LIN {X 0.012,Y -514.409,Z 331.146,A 0.000,B 0.000,C 90.000,E1 62.281} C_DIS
LIN {X 0.151,Y -518.654,Z 331.138,A 0.000,B 0.000,C 90.000,E1 60.795} C_DIS
LIN {X 0.232,Y -524.544,Z 331.127,A 0.000,B 0.000,C 90.000,E1 58.742} C_DIS
LIN {X -0.129,Y -529.522,Z 331.117,A 0.000,B 0.000,C 90.000,E1 57.041} C_DIS
LIN {X -0.088,Y -534.347,Z 331.107,A 0.000,B 0.000,C 90.000,E1 55.308} C_DIS
LIN {X 0.036,Y -537.358,Z 331.101,A 0.000,B 0.000,C 90.000,E1 54.149} C_DIS
LIN {X 0.091,Y -540.930,Z 331.093,A 0.000,B 0.000,C 90.000,E1 52.718} C_DIS
LIN {X -0.217,Y -544.110,Z 331.085,A 0.000,B 0.000,C 90.000,E1 51.331} C_DIS
LIN {X -0.125,Y -546.940,Z 331.077,A 0.000,B 0.000,C 90.000,E1 49.908} C_DIS
LIN {X 0.018,Y -549.384,Z 331.069,A 0.000,B 0.000,C 90.000,E1 48.485} C_DIS
LIN {X -0.259,Y -551.029,Z 331.063,A 0.000,B 0.000,C 90.000,E1 47.391} C_DIS
LIN {X -0.155,Y -552.114,Z 331.059,A 0.000,B 0.000,C 90.000,E1 46.539} C_DIS
LIN {X 0.343,Y -552.994,Z 331.054,A 0.000,B 0.000,C 90.000,E1 45.648} C_DIS
LIN {X 0.031,Y -553.500,Z 331.051,A 0.000,B 0.000,C 90.000,E1 45.121} C_DIS
LIN {X -0.195,Y -554.104,Z 331.045,A 0.000,B 0.000,C 90.000,E1 44.028} C_DIS
LIN {X -0.056,Y -554.318,Z 331.040,A 0.000,B 0.000,C 90.000,E1 43.176} C_DIS
LIN {X 0.110,Y -554.396,Z 331.034,A 0.000,B 0.000,C 90.000,E1 42.043} C_DIS
LIN {X -0.045,Y -553.917,Z 331.026,A 0.000,B 0.000,C 90.000,E1 40.663} C_DIS
LIN {X -0.209,Y -553.210,Z 331.020,A 0.000,B 0.000,C 90.000,E1 39.564} C_DIS
LIN {X 0.056,Y -552.229,Z 331.014,A 0.000,B 0.000,C 90.000,E1 38.418} C_DIS
LIN {X 0.062,Y -550.152,Z 331.003,A 0.000,B 0.000,C 90.000,E1 36.457} C_DIS
LIN {X 0.287,Y -548.915,Z 330.996,A 0.000,B 0.000,C 90.000,E1 35.311} C_DIS
LIN {X -0.221,Y -545.981,Z 330.982,A 0.000,B 0.000,C 90.000,E1 32.832} C_DIS
LIN {X 0.076,Y -543.685,Z 330.970,A 0.000,B 0.000,C 90.000,E1 30.541} C_DIS
LIN {X 0.017,Y -541.800,Z 330.959,A 0.000,B 0.000,C 90.000,E1 28.565} C_DIS
LIN {X 0.132,Y -539.961,Z 330.948,A 0.000,B 0.000,C 90.000,E1 26.565} C_DIS
LIN {X -0.042,Y -538.136,Z 330.937,A 0.000,B 0.000,C 90.000,E1 24.591} C_DIS
LIN {X 0.146,Y -535.740,Z 330.921,A 0.000,B 0.000,C 90.000,E1 21.716} C_DIS
LIN {X -0.070,Y -534.402,Z 330.908,A 0.000,B 0.000,C 90.000,E1 19.450} C_DIS
LIN {X 0.083,Y -533.648,Z 330.900,A 0.000,B 0.000,C 90.000,E1 18.000} C_DIS
LIN {X -0.002,Y -532.590,Z 330.886,A 0.000,B 0.000,C 90.000,E1 15.426} C_DIS
LIN {X 0.156,Y -531.870,Z 330.870,A 0.000,B 0.000,C 90.000,E1 12.535} C_DIS
LIN {X -0.064,Y -531.909,Z 330.859,A 0.000,B 0.000,C 90.000,E1 10.546} C_DIS
LIN {X 0.059,Y -532.143,Z 330.851,A 0.000,B 0.000,C 90.000,E1 9.095} C_DIS
LIN {X 0.283,Y -533.157,Z 330.833,A 0.000,B 0.000,C 90.000,E1 5.910} C_DIS
LIN {X -0.208,Y -534.755,Z 330.817,A 0.000,B 0.000,C 90.000,E1 3.094} C_DIS
LIN {X -0.196,Y -536.050,Z 330.808,A 0.000,B 0.000,C 90.000,E1 1.375} C_DIS
LIN {X 0.232,Y -538.074,Z 330.794,A 0.000,B 0.000,C 90.000,E1 358.912} C_DIS
LIN {X -0.140,Y -541.024,Z 330.780,A 0.000,B 0.000,C 90.000,E1 356.388} C_DIS
LIN {X -0.052,Y -542.072,Z 330.775,A 0.000,B 0.000,C 90.000,E1 355.527} C_DIS
LIN {X -0.243,Y -544.870,Z 330.763,A 0.000,B 0.000,C 90.000,E1 353.280} C_DIS
LIN {X -0.073,Y -550.293,Z 330.747,A 0.000,B 0.000,C 90.000,E1 350.443} C_DIS
LIN {X 0.094,Y -554.449,Z 330.736,A 0.000,B 0.000,C 90.000,E1 348.465} C_DIS
LIN {X 0.198,Y -558.087,Z 330.728,A 0.000,B 0.000,C 90.000,E1 347.061} C_DIS
LIN {X -0.196,Y -561.292,Z 330.722,A 0.000,B 0.000,C 90.000,E1 345.992} C_DIS
LIN {X -0.225,Y -565.993,Z 330.713,A 0.000,B 0.000,C 90.000,E1 344.338} C_DIS
LIN {X -0.212,Y -571.858,Z 330.702,A 0.000,B 0.000,C 90.000,E1 342.417} C_DIS
LIN {X -0.063,Y -576.026,Z 330.695,A 0.000,B 0.000,C 90.000,E1 341.040} C_DIS
LIN {X 0.156,Y -579.489,Z 330.689,A 0.000,B 0.000,C 90.000,E1 339.934} C_DIS
LIN {X 0.000,Y -586.299,Z 330.677,A 0.000,B 0.000,C 90.000,E1 337.794} C_DIS
LIN {X 0.140,Y -591.574,Z 330.668,A 0.000,B 0.000,C 90.000,E1 336.177} C_DIS
LIN {X 0.011,Y -598.007,Z 330.657,A 0.000,B 0.000,C 90.000,E1 334.332} C_DIS
LIN {X 0.172,Y -602.682,Z 330.650,A 0.000,B 0.000,C 90.000,E1 332.999} C_DIS
LIN {X 0.099,Y -608.216,Z 330.641,A 0.000,B 0.000,C 90.000,E1 331.435} C_DIS
LIN {X 0.103,Y -614.880,Z 330.631,A 0.000,B 0.000,C 90.000,E1 329.616} C_DIS
LIN {X 0.092,Y -618.751,Z 330.626,A 0.000,B 0.000,C 90.000,E1 328.584} C_DIS
LIN {X -0.186,Y -622.410,Z 330.620,A 0.000,B 0.000,C 90.000,E1 327.582} C_DIS
LIN {X -0.081,Y -625.914,Z 330.614,A 0.000,B 0.000,C 90.000,E1 326.548} C_DIS
LIN {X 0.072,Y -629.105,Z 330.608,A 0.000,B 0.000,C 90.000,E1 325.515} C_DIS
LIN {X -0.253,Y -632.881,Z 330.601,A 0.000,B 0.000,C 90.000,E1 324.276} C_DIS
LIN {X -0.157,Y -636.478,Z 330.594,A 0.000,B 0.000,C 90.000,E1 323.004} C_DIS
LIN {X 0.178,Y -642.080,Z 330.583,A 0.000,B 0.000,C 90.000,E1 320.964} C_DIS
LIN {X 0.162,Y -647.168,Z 330.574,A 0.000,B 0.000,C 90.000,E1 319.218} C_DIS
LIN {X -0.158,Y -651.503,Z 330.565,A 0.000,B 0.000,C 90.000,E1 317.757} C_DIS
LIN {X -0.002,Y -657.646,Z 330.554,A 0.000,B 0.000,C 90.000,E1 315.769} C_DIS
LIN {X 0.352,Y -660.733,Z 330.549,A 0.000,B 0.000,C 90.000,E1 314.757} C_DIS
LIN {X 0.263,Y -665.160,Z 330.541,A 0.000,B 0.000,C 90.000,E1 313.299} C_DIS
LIN {X 0.285,Y -669.342,Z 330.533,A 0.000,B 0.000,C 90.000,E1 311.838} C_DIS
LIN {X 0.379,Y -672.572,Z 330.526,A 0.000,B 0.000,C 90.000,E1 310.620} C_DIS
LIN {X 0.104,Y -676.131,Z 330.518,A 0.000,B 0.000,C 90.000,E1 309.197} C_DIS
LIN {X 0.254,Y -677.790,Z 330.514,A 0.000,B 0.000,C 90.000,E1 308.463} C_DIS
LIN {X 0.021,Y -679.783,Z 330.509,A 0.000,B 0.000,C 90.000,E1 307.523} C_DIS
LIN {X -0.187,Y -681.527,Z 330.503,A 0.000,B 0.000,C 90.000,E1 306.583} C_DIS
LIN {X 0.174,Y -682.972,Z 330.498,A 0.000,B 0.000,C 90.000,E1 305.598} C_DIS
LIN {X -0.007,Y -684.060,Z 330.493,A 0.000,B 0.000,C 90.000,E1 304.659} C_DIS
LIN {X -0.201,Y -684.530,Z 330.490,A 0.000,B 0.000,C 90.000,E1 304.199} C_DIS
LIN {X 0.189,Y -684.919,Z 330.486,A 0.000,B 0.000,C 90.000,E1 303.452} C_DIS
LIN {X 0.011,Y -685.079,Z 330.482,A 0.000,B 0.000,C 90.000,E1 302.752} C_DIS
LIN {X -0.172,Y -684.918,Z 330.478,A 0.000,B 0.000,C 90.000,E1 302.054} C_DIS
LIN {X 0.068,Y -684.319,Z 330.473,A 0.000,B 0.000,C 90.000,E1 301.082} C_DIS
LIN {X -0.136,Y -683.579,Z 330.469,A 0.000,B 0.000,C 90.000,E1 300.384} C_DIS
LIN {X -0.106,Y -682.543,Z 330.465,A 0.000,B 0.000,C 90.000,E1 299.667} C_DIS
LIN {X 0.122,Y -680.896,Z 330.460,A 0.000,B 0.000,C 90.000,E1 298.693} C_DIS
LIN {X 0.131,Y -679.393,Z 330.456,A 0.000,B 0.000,C 90.000,E1 297.975} C_DIS
LIN {X -0.094,Y -676.631,Z 330.449,A 0.000,B 0.000,C 90.000,E1 296.796} C_DIS
LIN {X -0.069,Y -673.699,Z 330.442,A 0.000,B 0.000,C 90.000,E1 295.591} C_DIS
LIN {X -0.088,Y -670.569,Z 330.435,A 0.000,B 0.000,C 90.000,E1 294.387} C_DIS
LIN {X 0.182,Y -667.241,Z 330.429,A 0.000,B 0.000,C 90.000,E1 293.153} C_DIS
LIN {X 0.063,Y -662.413,Z 330.419,A 0.000,B 0.000,C 90.000,E1 291.461} C_DIS
LIN {X -0.038,Y -657.821,Z 330.410,A 0.000,B 0.000,C 90.000,E1 289.758} C_DIS
LIN {X -0.114,Y -654.115,Z 330.402,A 0.000,B 0.000,C 90.000,E1 288.290} C_DIS
LIN {X -0.257,Y -648.922,Z 330.389,A 0.000,B 0.000,C 90.000,E1 286.079} C_DIS
LIN {X 0.199,Y -645.195,Z 330.380,A 0.000,B 0.000,C 90.000,E1 284.300} C_DIS
LIN {X -0.043,Y -639.443,Z 330.362,A 0.000,B 0.000,C 90.000,E1 281.074} C_DIS
LIN {X 0.336,Y -635.832,Z 330.346,A 0.000,B 0.000,C 90.000,E1 278.276} C_DIS
LIN {X 0.019,Y -633.257,Z 330.329,A 0.000,B 0.000,C 90.000,E1 275.277} C_DIS
LIN {X -0.167,Y -631.822,Z 330.311,A 0.000,B 0.000,C 90.000,E1 272.007} C_DIS
LIN {X -0.008,Y -631.589,Z 330.298,A 0.000,B 0.000,C 90.000,E1 269.714} C_DIS
LIN {X 0.147,Y -632.009,Z 330.286,A 0.000,B 0.000,C 90.000,E1 267.421} C_DIS
LIN {X 0.246,Y -632.814,Z 330.276,A 0.000,B 0.000,C 90.000,E1 265.641} C_DIS
LIN {X -0.211,Y -633.900,Z 330.266,A 0.000,B 0.000,C 90.000,E1 263.913} C_DIS
LIN {X 0.258,Y -635.065,Z 330.258,A 0.000,B 0.000,C 90.000,E1 262.356} C_DIS
LIN {X -0.263,Y -636.792,Z 330.247,A 0.000,B 0.000,C 90.000,E1 260.387} C_DIS
LIN {X 0.114,Y -638.970,Z 330.235,A 0.000,B 0.000,C 90.000,E1 258.342} C_DIS
LIN {X 0.081,Y -641.221,Z 330.226,A 0.000,B 0.000,C 90.000,E1 256.589} C_DIS
LIN {X 0.072,Y -642.543,Z 330.220,A 0.000,B 0.000,C 90.000,E1 255.589} C_DIS
LIN {X -0.227,Y -643.320,Z 330.216,A 0.000,B 0.000,C 90.000,E1 254.866} C_DIS
LIN {X -0.186,Y -644.381,Z 330.209,A 0.000,B 0.000,C 90.000,E1 253.614} C_DIS
LIN {X -0.133,Y -645.125,Z 330.202,A 0.000,B 0.000,C 90.000,E1 252.362} C_DIS
LIN {X 0.223,Y -645.400,Z 330.198,A 0.000,B 0.000,C 90.000,E1 251.583} C_DIS
LIN {X -0.033,Y -645.324,Z 330.194,A 0.000,B 0.000,C 90.000,E1 250.859} C_DIS
LIN {X 0.024,Y -645.305,Z 330.192,A 0.000,B 0.000,C 90.000,E1 250.604} C_DIS
LIN {X -0.232,Y -644.846,Z 330.188,A 0.000,B 0.000,C 90.000,E1 249.880} C_DIS
LIN {X -0.332,Y -644.440,Z 330.185,A 0.000,B 0.000,C 90.000,E1 249.390} C_DIS
LIN {X 0.229,Y -643.507,Z 330.181,A 0.000,B 0.000,C 90.000,E1 248.592} C_DIS
LIN {X 0.118,Y -642.776,Z 330.178,A 0.000,B 0.000,C 90.000,E1 248.103} C_DIS
LIN {X 0.064,Y -641.430,Z 330.174,A 0.000,B 0.000,C 90.000,E1 247.358} C_DIS
LIN {X -0.064,Y -640.421,Z 330.172,A 0.000,B 0.000,C 90.000,E1 246.869} C_DIS
LIN {X -0.090,Y -638.024,Z 330.166,A 0.000,B 0.000,C 90.000,E1 245.869} C_DIS
LIN {X 0.069,Y -636.071,Z 330.162,A 0.000,B 0.000,C 90.000,E1 245.101} C_DIS
LIN {X 0.167,Y -634.684,Z 330.159,A 0.000,B 0.000,C 90.000,E1 244.588} C_DIS
LIN {X 0.059,Y -631.483,Z 330.153,A 0.000,B 0.000,C 90.000,E1 243.589} C_DIS
LIN {X 0.179,Y -628.105,Z 330.148,A 0.000,B 0.000,C 90.000,E1 242.564} C_DIS
LIN {X 0.007,Y -623.774,Z 330.141,A 0.000,B 0.000,C 90.000,E1 241.307} C_DIS
LIN {X 0.015,Y -620.333,Z 330.135,A 0.000,B 0.000,C 90.000,E1 240.284} C_DIS
LIN {X 0.010,Y -615.064,Z 330.126,A 0.000,B 0.000,C 90.000,E1 238.742} C_DIS
LIN {X 0.231,Y -609.789,Z 330.118,A 0.000,B 0.000,C 90.000,E1 237.168} C_DIS
LIN {X 0.082,Y -605.275,Z 330.111,A 0.000,B 0.000,C 90.000,E1 235.881} C_DIS
LIN {X 0.083,Y -597.989,Z 330.099,A 0.000,B 0.000,C 90.000,E1 233.783} C_DIS
LIN {X -0.292,Y -594.305,Z 330.093,A 0.000,B 0.000,C 90.000,E1 232.763} C_DIS
LIN {X 0.108,Y -586.649,Z 330.081,A 0.000,B 0.000,C 90.000,E1 230.598} C_DIS
LIN {X 0.131,Y -582.072,Z 330.074,A 0.000,B 0.000,C 90.000,E1 229.256} C_DIS
LIN {X 0.029,Y -574.882,Z 330.062,A 0.000,B 0.000,C 90.000,E1 227.106} C_DIS
LIN {X 0.197,Y -570.377,Z 330.054,A 0.000,B 0.000,C 90.000,E1 225.729} C_DIS
LIN {X -0.018,Y -565.003,Z 330.045,A 0.000,B 0.000,C 90.000,E1 224.109} C_DIS
LIN {X 0.140,Y -558.793,Z 330.034,A 0.000,B 0.000,C 90.000,E1 222.162} C_DIS
LIN {X -0.225,Y -552.620,Z 330.024,A 0.000,B 0.000,C 90.000,E1 220.253} C_DIS
LIN {X 0.053,Y -547.411,Z 330.014,A 0.000,B 0.000,C 90.000,E1 218.543} C_DIS
LIN {X -0.096,Y -541.470,Z 330.003,A 0.000,B 0.000,C 90.000,E1 216.583} C_DIS
LIN {X 0.168,Y -535.054,Z 329.991,A 0.000,B 0.000,C 90.000,E1 214.278} C_DIS
LIN {X -0.052,Y -529.022,Z 329.978,A 0.000,B 0.000,C 90.000,E1 212.005} C_DIS
LIN {X -0.233,Y -524.175,Z 329.967,A 0.000,B 0.000,C 90.000,E1 210.001} C_DIS
LIN {X -0.078,Y -521.442,Z 329.960,A 0.000,B 0.000,C 90.000,E1 208.821} C_DIS
LIN {X 0.200,Y -516.746,Z 329.949,A 0.000,B 0.000,C 90.000,E1 206.744} C_DIS
LIN {X 0.123,Y -513.496,Z 329.941,A 0.000,B 0.000,C 90.000,E1 205.283} C_DIS
LIN {X -0.126,Y -510.935,Z 329.934,A 0.000,B 0.000,C 90.000,E1 204.131} C_DIS
LIN {X -0.055,Y -507.615,Z 329.926,A 0.000,B 0.000,C 90.000,E1 202.642} C_DIS
LIN {X -0.052,Y -502.946,Z 329.914,A 0.000,B 0.000,C 90.000,E1 200.556} C_DIS
LIN {X 0.233,Y -498.998,Z 329.904,A 0.000,B 0.000,C 90.000,E1 198.725} C_DIS
LIN {X 0.258,Y -495.156,Z 329.894,A 0.000,B 0.000,C 90.000,E1 196.913} C_DIS
LIN {X -0.085,Y -491.558,Z 329.884,A 0.000,B 0.000,C 90.000,E1 195.134} C_DIS
LIN {X -0.023,Y -488.185,Z 329.874,A 0.000,B 0.000,C 90.000,E1 193.300} C_DIS
LIN {X -0.030,Y -485.458,Z 329.865,A 0.000,B 0.000,C 90.000,E1 191.771} C_DIS
LIN {X -0.188,Y -482.775,Z 329.857,A 0.000,B 0.000,C 90.000,E1 190.254} C_DIS
LIN {X -0.145,Y -479.614,Z 329.847,A 0.000,B 0.000,C 90.000,E1 188.398} C_DIS
LIN {X -0.090,Y -475.772,Z 329.833,A 0.000,B 0.000,C 90.000,E1 185.910} C_DIS
LIN {X 0.177,Y -472.347,Z 329.819,A 0.000,B 0.000,C 90.000,E1 183.383} C_DIS
LIN {X -0.153,Y -469.340,Z 329.805,A 0.000,B 0.000,C 90.000,E1 180.917} C_DIS
LIN {X -0.126,Y -467.003,Z 329.791,A 0.000,B 0.000,C 90.000,E1 178.396} C_DIS
LIN {X 0.107,Y -464.884,Z 329.772,A 0.000,B 0.000,C 90.000,E1 174.894} C_DIS
LIN {X -0.050,Y -464.115,Z 329.756,A 0.000,B 0.000,C 90.000,E1 172.064} C_DIS
LIN {X -0.148,Y -464.067,Z 329.744,A 0.000,B 0.000,C 90.000,E1 169.859} C_DIS
LIN {X 0.200,Y -465.056,Z 329.721,A 0.000,B 0.000,C 90.000,E1 165.700} C_DIS
LIN {X 0.061,Y -466.232,Z 329.708,A 0.000,B 0.000,C 90.000,E1 163.504} C_DIS
LIN {X 0.191,Y -469.670,Z 329.686,A 0.000,B 0.000,C 90.000,E1 159.390} C_DIS
LIN {X -0.222,Y -473.534,Z 329.668,A 0.000,B 0.000,C 90.000,E1 156.305} C_DIS
LIN {X 0.131,Y -477.489,Z 329.654,A 0.000,B 0.000,C 90.000,E1 153.768} C_DIS
LIN {X -0.019,Y -482.266,Z 329.641,A 0.000,B 0.000,C 90.000,E1 151.307} C_DIS
LIN {X -0.031,Y -486.993,Z 329.629,A 0.000,B 0.000,C 90.000,E1 149.154} C_DIS
LIN {X 0.089,Y -489.890,Z 329.622,A 0.000,B 0.000,C 90.000,E1 147.916} C_DIS
LIN {X -0.002,Y -493.123,Z 329.615,A 0.000,B 0.000,C 90.000,E1 146.707} C_DIS
LIN {X -0.191,Y -498.875,Z 329.603,A 0.000,B 0.000,C 90.000,E1 144.609} C_DIS
LIN {X 0.180,Y -503.920,Z 329.593,A 0.000,B 0.000,C 90.000,E1 142.763} C_DIS
LIN {X -0.255,Y -507.135,Z 329.587,A 0.000,B 0.000,C 90.000,E1 141.618} C_DIS
LIN {X -0.237,Y -509.324,Z 329.582,A 0.000,B 0.000,C 90.000,E1 140.723} C_DIS
LIN {X -0.192,Y -511.355,Z 329.577,A 0.000,B 0.000,C 90.000,E1 139.828} C_DIS
LIN {X 0.041,Y -514.326,Z 329.569,A 0.000,B 0.000,C 90.000,E1 138.324} C_DIS
LIN {X -0.248,Y -515.862,Z 329.564,A 0.000,B 0.000,C 90.000,E1 137.472} C_DIS
LIN {X 0.209,Y -517.062,Z 329.559,A 0.000,B 0.000,C 90.000,E1 136.539} C_DIS
LIN {X 0.305,Y -517.835,Z 329.554,A 0.000,B 0.000,C 90.000,E1 135.648} C_DIS
LIN {X -0.038,Y -518.443,Z 329.547,A 0.000,B 0.000,C 90.000,E1 134.514} C_DIS
LIN {X 0.075,Y -518.571,Z 329.542,A 0.000,B 0.000,C 90.000,E1 133.623} C_DIS
LIN {X -0.097,Y -518.502,Z 329.539,A 0.000,B 0.000,C 90.000,E1 133.056} C_DIS
LIN {X 0.042,Y -518.148,Z 329.534,A 0.000,B 0.000,C 90.000,E1 132.162} C_DIS
LIN {X -0.204,Y -517.471,Z 329.529,A 0.000,B 0.000,C 90.000,E1 131.310} C_DIS
LIN {X -0.066,Y -516.523,Z 329.525,A 0.000,B 0.000,C 90.000,E1 130.415} C_DIS
LIN {X 0.320,Y -515.023,Z 329.518,A 0.000,B 0.000,C 90.000,E1 129.197} C_DIS
LIN {X 0.199,Y -512.590,Z 329.508,A 0.000,B 0.000,C 90.000,E1 127.443} C_DIS
LIN {X -0.120,Y -510.914,Z 329.502,A 0.000,B 0.000,C 90.000,E1 126.297} C_DIS
LIN {X -0.049,Y -509.074,Z 329.495,A 0.000,B 0.000,C 90.000,E1 125.105} C_DIS
LIN {X -0.008,Y -506.958,Z 329.488,A 0.000,B 0.000,C 90.000,E1 123.913} C_DIS
LIN {X 0.034,Y -504.105,Z 329.480,A 0.000,B 0.000,C 90.000,E1 122.418} C_DIS
LIN {X -0.157,Y -502.292,Z 329.475,A 0.000,B 0.000,C 90.000,E1 121.544} C_DIS
LIN {X -0.167,Y -498.590,Z 329.465,A 0.000,B 0.000,C 90.000,E1 119.745} C_DIS
LIN {X -0.108,Y -495.312,Z 329.457,A 0.000,B 0.000,C 90.000,E1 118.231} C_DIS
LIN {X -0.066,Y -490.773,Z 329.445,A 0.000,B 0.000,C 90.000,E1 116.104} C_DIS
LIN {X -0.165,Y -487.434,Z 329.437,A 0.000,B 0.000,C 90.000,E1 114.591} C_DIS
LIN {X 0.121,Y -483.973,Z 329.428,A 0.000,B 0.000,C 90.000,E1 113.025} C_DIS
LIN {X 0.151,Y -479.763,Z 329.418,A 0.000,B 0.000,C 90.000,E1 111.173} C_DIS
LIN {X 0.128,Y -477.600,Z 329.413,A 0.000,B 0.000,C 90.000,E1 110.248} C_DIS
LIN {X -0.134,Y -473.705,Z 329.404,A 0.000,B 0.000,C 90.000,E1 108.725} C_DIS
LIN {X 0.019,Y -470.581,Z 329.397,A 0.000,B 0.000,C 90.000,E1 107.457} C_DIS
LIN {X -0.016,Y -467.271,Z 329.390,A 0.000,B 0.000,C 90.000,E1 106.205} C_DIS
LIN {X 0.118,Y -465.868,Z 329.387,A 0.000,B 0.000,C 90.000,E1 105.662} C_DIS
LIN {X 0.078,Y -465.863,Z 329.387,A 0.000,B 0.000,C 90.000,E1 105.662} C_DIS
LIN {X -0.099,Y -467.672,Z 329.383,A 0.000,B 0.000,C 90.000,E1 104.954} C_DIS
LIN {X -0.141,Y -475.886,Z 329.357,A 0.000,B 0.000,C 90.000,E1 100.254} C_DIS
LIN {X 0.166,Y -476.343,Z 329.355,A 0.000,B 0.000,C 90.000,E1 99.905} C_DIS
LIN {X 0.123,Y -481.853,Z 329.331,A 0.000,B 0.000,C 90.000,E1 95.568} C_DIS
LIN {X -0.031,Y -482.187,Z 329.329,A 0.000,B 0.000,C 90.000,E1 95.277} C_DIS
LIN {X -0.097,Y -485.350,Z 329.305,A 0.000,B 0.000,C 90.000,E1 90.974} C_DIS
LIN {X 0.213,Y -485.533,Z 329.304,A 0.000,B 0.000,C 90.000,E1 90.630} C_DIS
LIN {X -0.065,Y -486.339,Z 329.282,A 0.000,B 0.000,C 90.000,E1 86.674} C_DIS
LIN {X 0.069,Y -486.277,Z 329.278,A 0.000,B 0.000,C 90.000,E1 86.045} C_DIS
LIN {X -0.211,Y -484.694,Z 329.254,A 0.000,B 0.000,C 90.000,E1 81.781} C_DIS
LIN {X 0.137,Y -484.551,Z 329.253,A 0.000,B 0.000,C 90.000,E1 81.432} C_DIS
LIN {X 0.007,Y -480.491,Z 329.227,A 0.000,B 0.000,C 90.000,E1 76.825} C_DIS
LIN {X 0.206,Y -477.337,Z 329.215,A 0.000,B 0.000,C 90.000,E1 74.755} C_DIS
LIN {X 0.166,Y -477.338,Z 329.215,A 0.000,B 0.000,C 90.000,E1 74.755} C_DIS
LIN {X -0.103,Y -480.709,Z 329.210,A 0.000,B 0.000,C 90.000,E1 73.740} C_DIS
LIN {X 0.178,Y -483.615,Z 329.204,A 0.000,B 0.000,C 90.000,E1 72.779} C_DIS
LIN {X -0.100,Y -487.983,Z 329.196,A 0.000,B 0.000,C 90.000,E1 71.275} C_DIS
LIN {X -0.140,Y -492.281,Z 329.187,A 0.000,B 0.000,C 90.000,E1 69.752} C_DIS
LIN {X -0.104,Y -496.633,Z 329.179,A 0.000,B 0.000,C 90.000,E1 68.230} C_DIS
LIN {X 0.125,Y -500.116,Z 329.172,A 0.000,B 0.000,C 90.000,E1 66.997} C_DIS
LIN {X -0.075,Y -506.113,Z 329.161,A 0.000,B 0.000,C 90.000,E1 64.921} C_DIS
LIN {X 0.002,Y -511.279,Z 329.151,A 0.000,B 0.000,C 90.000,E1 63.127} C_DIS
LIN {X -0.264,Y -516.377,Z 329.141,A 0.000,B 0.000,C 90.000,E1 61.385} C_DIS
LIN {X 0.157,Y -520.579,Z 329.133,A 0.000,B 0.000,C 90.000,E1 59.871} C_DIS
LIN {X 0.208,Y -524.782,Z 329.125,A 0.000,B 0.000,C 90.000,E1 58.408} C_DIS
LIN {X -0.149,Y -529.790,Z 329.115,A 0.000,B 0.000,C 90.000,E1 56.707} C_DIS
LIN {X -0.099,Y -533.800,Z 329.107,A 0.000,B 0.000,C 90.000,E1 55.261} C_DIS
LIN {X -0.110,Y -536.848,Z 329.101,A 0.000,B 0.000,C 90.000,E1 54.116} C_DIS
LIN {X -0.070,Y -539.716,Z 329.094,A 0.000,B 0.000,C 90.000,E1 52.970} C_DIS
LIN {X 0.036,Y -542.959,Z 329.086,A 0.000,B 0.000,C 90.000,E1 51.537} C_DIS
LIN {X -0.269,Y -545.289,Z 329.080,A 0.000,B 0.000,C 90.000,E1 50.436} C_DIS
LIN {X 0.184,Y -546.922,Z 329.075,A 0.000,B 0.000,C 90.000,E1 49.542} C_DIS
LIN {X -0.126,Y -548.880,Z 329.069,A 0.000,B 0.000,C 90.000,E1 48.447} C_DIS
LIN {X 0.002,Y -550.532,Z 329.063,A 0.000,B 0.000,C 90.000,E1 47.310} C_DIS
LIN {X 0.102,Y -551.631,Z 329.058,A 0.000,B 0.000,C 90.000,E1 46.458} C_DIS
LIN {X -0.187,Y -552.538,Z 329.054,A 0.000,B 0.000,C 90.000,E1 45.648} C_DIS
LIN {X -0.074,Y -553.249,Z 329.049,A 0.000,B 0.000,C 90.000,E1 44.798} C_DIS
LIN {X 0.048,Y -553.721,Z 329.044,A 0.000,B 0.000,C 90.000,E1 43.947} C_DIS
LIN {X 0.182,Y -553.999,Z 329.040,A 0.000,B 0.000,C 90.000,E1 43.095} C_DIS
LIN {X -0.026,Y -554.142,Z 329.033,A 0.000,B 0.000,C 90.000,E1 42.000} C_DIS
LIN {X 0.178,Y -553.931,Z 329.027,A 0.000,B 0.000,C 90.000,E1 40.862} C_DIS
LIN {X 0.312,Y -553.581,Z 329.023,A 0.000,B 0.000,C 90.000,E1 40.011} C_DIS
LIN {X 0.149,Y -552.782,Z 329.016,A 0.000,B 0.000,C 90.000,E1 38.910} C_DIS
LIN {X -0.087,Y -552.007,Z 329.012,A 0.000,B 0.000,C 90.000,E1 38.096} C_DIS
LIN {X -0.157,Y -550.296,Z 329.002,A 0.000,B 0.000,C 90.000,E1 36.423} C_DIS
LIN {X -0.256,Y -549.056,Z 328.996,A 0.000,B 0.000,C 90.000,E1 35.311} C_DIS
LIN {X -0.002,Y -546.142,Z 328.982,A 0.000,B 0.000,C 90.000,E1 32.752} C_DIS
LIN {X 0.292,Y -543.860,Z 328.969,A 0.000,B 0.000,C 90.000,E1 30.463} C_DIS
LIN {X 0.230,Y -541.988,Z 328.958,A 0.000,B 0.000,C 90.000,E1 28.487} C_DIS
LIN {X -0.142,Y -540.147,Z 328.947,A 0.000,B 0.000,C 90.000,E1 26.539} C_DIS
LIN {X 0.163,Y -538.318,Z 328.936,A 0.000,B 0.000,C 90.000,E1 24.515} C_DIS
LIN {X 0.144,Y -535.937,Z 328.920,A 0.000,B 0.000,C 90.000,E1 21.663} C_DIS
LIN {X -0.084,Y -534.755,Z 328.909,A 0.000,B 0.000,C 90.000,E1 19.685} C_DIS
LIN {X 0.102,Y -533.848,Z 328.900,A 0.000,B 0.000,C 90.000,E1 17.946} C_DIS
LIN {X 0.031,Y -532.786,Z 328.885,A 0.000,B 0.000,C 90.000,E1 15.371} C_DIS
LIN {X 0.202,Y -532.082,Z 328.870,A 0.000,B 0.000,C 90.000,E1 12.479} C_DIS
LIN {X -0.009,Y -532.119,Z 328.858,A 0.000,B 0.000,C 90.000,E1 10.489} C_DIS
LIN {X 0.204,Y -532.355,Z 328.850,A 0.000,B 0.000,C 90.000,E1 9.029} C_DIS
LIN {X -0.210,Y -533.275,Z 328.834,A 0.000,B 0.000,C 90.000,E1 6.201} C_DIS
LIN {X -0.124,Y -534.985,Z 328.817,A 0.000,B 0.000,C 90.000,E1 3.037} C_DIS
LIN {X -0.102,Y -536.507,Z 328.806,A 0.000,B 0.000,C 90.000,E1 1.031} C_DIS
LIN {X -0.211,Y -540.025,Z 328.785,A 0.000,B 0.000,C 90.000,E1 357.249} C_DIS
LIN {X -0.048,Y -542.041,Z 328.775,A 0.000,B 0.000,C 90.000,E1 355.527} C_DIS
LIN {X -0.158,Y -545.172,Z 328.761,A 0.000,B 0.000,C 90.000,E1 352.989} C_DIS
LIN {X -0.077,Y -550.039,Z 328.747,A 0.000,B 0.000,C 90.000,E1 350.443} C_DIS
LIN {X 0.208,Y -554.848,Z 328.734,A 0.000,B 0.000,C 90.000,E1 348.173} C_DIS
LIN {X 0.182,Y -557.700,Z 328.728,A 0.000,B 0.000,C 90.000,E1 347.061} C_DIS
LIN {X 0.183,Y -560.145,Z 328.724,A 0.000,B 0.000,C 90.000,E1 346.228} C_DIS
LIN {X 0.059,Y -566.428,Z 328.711,A 0.000,B 0.000,C 90.000,E1 344.031} C_DIS
LIN {X 0.293,Y -571.413,Z 328.702,A 0.000,B 0.000,C 90.000,E1 342.362} C_DIS
LIN {X -0.109,Y -575.583,Z 328.695,A 0.000,B 0.000,C 90.000,E1 341.040} C_DIS
LIN {X -0.258,Y -579.814,Z 328.687,A 0.000,B 0.000,C 90.000,E1 339.699} C_DIS
LIN {X 0.097,Y -588.430,Z 328.672,A 0.000,B 0.000,C 90.000,E1 336.975} C_DIS
LIN {X 0.006,Y -596.584,Z 328.659,A 0.000,B 0.000,C 90.000,E1 334.588} C_DIS
LIN {X 0.141,Y -601.287,Z 328.652,A 0.000,B 0.000,C 90.000,E1 333.256} C_DIS
LIN {X -0.065,Y -604.086,Z 328.647,A 0.000,B 0.000,C 90.000,E1 332.487} C_DIS
LIN {X -0.160,Y -610.567,Z 328.637,A 0.000,B 0.000,C 90.000,E1 330.667} C_DIS
LIN {X 0.256,Y -615.401,Z 328.630,A 0.000,B 0.000,C 90.000,E1 329.331} C_DIS
LIN {X -0.064,Y -619.250,Z 328.624,A 0.000,B 0.000,C 90.000,E1 328.329} C_DIS
LIN {X -0.005,Y -622.834,Z 328.618,A 0.000,B 0.000,C 90.000,E1 327.296} C_DIS
LIN {X 0.295,Y -625.460,Z 328.614,A 0.000,B 0.000,C 90.000,E1 326.501} C_DIS
LIN {X -0.087,Y -629.421,Z 328.607,A 0.000,B 0.000,C 90.000,E1 325.261} C_DIS
LIN {X -0.046,Y -633.157,Z 328.600,A 0.000,B 0.000,C 90.000,E1 323.989} C_DIS
LIN {X 0.057,Y -636.018,Z 328.594,A 0.000,B 0.000,C 90.000,E1 322.970} C_DIS
LIN {X -0.003,Y -640.931,Z 328.585,A 0.000,B 0.000,C 90.000,E1 321.215} C_DIS
LIN {X -0.032,Y -646.699,Z 328.573,A 0.000,B 0.000,C 90.000,E1 319.218} C_DIS
LIN {X -0.305,Y -650.323,Z 328.567,A 0.000,B 0.000,C 90.000,E1 318.000} C_DIS
LIN {X 0.238,Y -657.144,Z 328.554,A 0.000,B 0.000,C 90.000,E1 315.729} C_DIS
LIN {X 0.126,Y -660.231,Z 328.549,A 0.000,B 0.000,C 90.000,E1 314.757} C_DIS
LIN {X 0.025,Y -664.624,Z 328.541,A 0.000,B 0.000,C 90.000,E1 313.299} C_DIS
LIN {X 0.035,Y -668.772,Z 328.533,A 0.000,B 0.000,C 90.000,E1 311.838} C_DIS
LIN {X 0.118,Y -671.947,Z 328.526,A 0.000,B 0.000,C 90.000,E1 310.620} C_DIS
LIN {X -0.170,Y -675.435,Z 328.518,A 0.000,B 0.000,C 90.000,E1 309.197} C_DIS
LIN {X -0.029,Y -677.057,Z 328.514,A 0.000,B 0.000,C 90.000,E1 308.463} C_DIS
LIN {X 0.284,Y -679.487,Z 328.507,A 0.000,B 0.000,C 90.000,E1 307.237} C_DIS
LIN {X 0.071,Y -681.117,Z 328.502,A 0.000,B 0.000,C 90.000,E1 306.297} C_DIS
LIN {X -0.140,Y -682.177,Z 328.498,A 0.000,B 0.000,C 90.000,E1 305.598} C_DIS
LIN {X -0.340,Y -682.973,Z 328.494,A 0.000,B 0.000,C 90.000,E1 304.898} C_DIS
LIN {X 0.417,Y -683.609,Z 328.490,A 0.000,B 0.000,C 90.000,E1 304.119} C_DIS
LIN {X -0.154,Y -684.005,Z 328.484,A 0.000,B 0.000,C 90.000,E1 303.214} C_DIS
LIN {X -0.338,Y -684.067,Z 328.482,A 0.000,B 0.000,C 90.000,E1 302.752} C_DIS
LIN {X -0.151,Y -684.005,Z 328.479,A 0.000,B 0.000,C 90.000,E1 302.260} C_DIS
LIN {X 0.431,Y -683.409,Z 328.474,A 0.000,B 0.000,C 90.000,E1 301.258} C_DIS
LIN {X -0.132,Y -682.737,Z 328.470,A 0.000,B 0.000,C 90.000,E1 300.590} C_DIS
LIN {X 0.094,Y -681.380,Z 328.465,A 0.000,B 0.000,C 90.000,E1 299.617} C_DIS
LIN {X 0.110,Y -680.120,Z 328.461,A 0.000,B 0.000,C 90.000,E1 298.899} C_DIS
LIN {X -0.286,Y -678.136,Z 328.455,A 0.000,B 0.000,C 90.000,E1 297.975} C_DIS
LIN {X 0.074,Y -675.355,Z 328.449,A 0.000,B 0.000,C 90.000,E1 296.744} C_DIS
LIN {X 0.084,Y -672.367,Z 328.442,A 0.000,B 0.000,C 90.000,E1 295.540} C_DIS
LIN {X 0.210,Y -668.566,Z 328.434,A 0.000,B 0.000,C 90.000,E1 294.079} C_DIS
LIN {X -0.163,Y -665.175,Z 328.427,A 0.000,B 0.000,C 90.000,E1 292.898} C_DIS
LIN {X 0.157,Y -661.049,Z 328.419,A 0.000,B 0.000,C 90.000,E1 291.408} C_DIS
LIN {X 0.032,Y -656.461,Z 328.410,A 0.000,B 0.000,C 90.000,E1 289.704} C_DIS
LIN {X -0.193,Y -652.157,Z 328.400,A 0.000,B 0.000,C 90.000,E1 288.000} C_DIS
LIN {X -0.240,Y -647.587,Z 328.389,A 0.000,B 0.000,C 90.000,E1 286.024} C_DIS
LIN {X -0.259,Y -642.409,Z 328.375,A 0.000,B 0.000,C 90.000,E1 283.536} C_DIS
LIN {X 0.015,Y -637.091,Z 328.357,A 0.000,B 0.000,C 90.000,E1 280.254} C_DIS
LIN {X -0.137,Y -632.935,Z 328.336,A 0.000,B 0.000,C 90.000,E1 276.486} C_DIS
LIN {X 0.098,Y -631.421,Z 328.323,A 0.000,B 0.000,C 90.000,E1 274.188} C_DIS
LIN {X 0.269,Y -630.607,Z 328.311,A 0.000,B 0.000,C 90.000,E1 271.892} C_DIS
LIN {X -0.239,Y -630.394,Z 328.298,A 0.000,B 0.000,C 90.000,E1 269.656} C_DIS
LIN {X -0.120,Y -630.849,Z 328.285,A 0.000,B 0.000,C 90.000,E1 267.364} C_DIS
LIN {X -0.323,Y -631.834,Z 328.274,A 0.000,B 0.000,C 90.000,E1 265.355} C_DIS
LIN {X -0.183,Y -632.982,Z 328.264,A 0.000,B 0.000,C 90.000,E1 263.571} C_DIS
LIN {X 0.342,Y -634.210,Z 328.256,A 0.000,B 0.000,C 90.000,E1 262.008} C_DIS
LIN {X -0.016,Y -635.789,Z 328.246,A 0.000,B 0.000,C 90.000,E1 260.274} C_DIS
LIN {X -0.126,Y -637.726,Z 328.236,A 0.000,B 0.000,C 90.000,E1 258.522} C_DIS
LIN {X -0.047,Y -640.000,Z 328.226,A 0.000,B 0.000,C 90.000,E1 256.756} C_DIS
LIN {X -0.223,Y -641.661,Z 328.219,A 0.000,B 0.000,C 90.000,E1 255.519} C_DIS
LIN {X -0.228,Y -642.720,Z 328.214,A 0.000,B 0.000,C 90.000,E1 254.519} C_DIS
LIN {X -0.052,Y -643.574,Z 328.208,A 0.000,B 0.000,C 90.000,E1 253.504} C_DIS
LIN {X 0.175,Y -644.386,Z 328.201,A 0.000,B 0.000,C 90.000,E1 252.236} C_DIS
LIN {X -0.133,Y -644.663,Z 328.199,A 0.000,B 0.000,C 90.000,E1 251.764} C_DIS
LIN {X 0.265,Y -644.674,Z 328.193,A 0.000,B 0.000,C 90.000,E1 250.732} C_DIS
LIN {X 0.106,Y -644.667,Z 328.192,A 0.000,B 0.000,C 90.000,E1 250.496} C_DIS
LIN {X -0.103,Y -644.105,Z 328.186,A 0.000,B 0.000,C 90.000,E1 249.518} C_DIS
LIN {X -0.209,Y -643.656,Z 328.183,A 0.000,B 0.000,C 90.000,E1 249.028} C_DIS
LIN {X -0.256,Y -642.787,Z 328.179,A 0.000,B 0.000,C 90.000,E1 248.284} C_DIS
LIN {X -0.370,Y -642.034,Z 328.177,A 0.000,B 0.000,C 90.000,E1 247.794} C_DIS
LIN {X 0.158,Y -640.673,Z 328.172,A 0.000,B 0.000,C 90.000,E1 246.997} C_DIS
LIN {X 0.277,Y -639.621,Z 328.170,A 0.000,B 0.000,C 90.000,E1 246.485} C_DIS
LIN {X 0.189,Y -637.822,Z 328.165,A 0.000,B 0.000,C 90.000,E1 245.741} C_DIS
LIN {X 0.396,Y -635.171,Z 328.160,A 0.000,B 0.000,C 90.000,E1 244.717} C_DIS
LIN {X -0.274,Y -632.042,Z 328.154,A 0.000,B 0.000,C 90.000,E1 243.768} C_DIS
LIN {X -0.139,Y -628.709,Z 328.149,A 0.000,B 0.000,C 90.000,E1 242.743} C_DIS
LIN {X -0.055,Y -625.308,Z 328.143,A 0.000,B 0.000,C 90.000,E1 241.719} C_DIS
LIN {X -0.269,Y -620.164,Z 328.134,A 0.000,B 0.000,C 90.000,E1 240.205} C_DIS
LIN {X -0.269,Y -614.975,Z 328.126,A 0.000,B 0.000,C 90.000,E1 238.663} C_DIS
LIN {X 0.191,Y -610.649,Z 328.119,A 0.000,B 0.000,C 90.000,E1 237.327} C_DIS
LIN {X 0.119,Y -607.153,Z 328.113,A 0.000,B 0.000,C 90.000,E1 236.294} C_DIS
LIN {X -0.074,Y -600.861,Z 328.103,A 0.000,B 0.000,C 90.000,E1 234.482} C_DIS
LIN {X 0.068,Y -597.290,Z 328.097,A 0.000,B 0.000,C 90.000,E1 233.417} C_DIS
LIN {X 0.157,Y -593.526,Z 328.091,A 0.000,B 0.000,C 90.000,E1 232.351} C_DIS
LIN {X -0.011,Y -584.202,Z 328.076,A 0.000,B 0.000,C 90.000,E1 229.703} C_DIS
LIN {X -0.326,Y -576.122,Z 328.063,A 0.000,B 0.000,C 90.000,E1 227.310} C_DIS
LIN {X 0.285,Y -571.690,Z 328.055,A 0.000,B 0.000,C 90.000,E1 225.891} C_DIS
LIN {X -0.213,Y -565.387,Z 328.045,A 0.000,B 0.000,C 90.000,E1 224.028} C_DIS
LIN {X -0.128,Y -560.106,Z 328.035,A 0.000,B 0.000,C 90.000,E1 222.366} C_DIS
LIN {X -0.117,Y -554.864,Z 328.026,A 0.000,B 0.000,C 90.000,E1 220.701} C_DIS
LIN {X 0.209,Y -549.633,Z 328.017,A 0.000,B 0.000,C 90.000,E1 218.991} C_DIS
LIN {X -0.010,Y -546.231,Z 328.011,A 0.000,B 0.000,C 90.000,E1 217.890} C_DIS
LIN {X -0.192,Y -540.338,Z 328.000,A 0.000,B 0.000,C 90.000,E1 215.931} C_DIS
LIN {X 0.030,Y -534.070,Z 327.987,A 0.000,B 0.000,C 90.000,E1 213.627} C_DIS
LIN {X -0.097,Y -527.439,Z 327.973,A 0.000,B 0.000,C 90.000,E1 211.052} C_DIS
LIN {X 0.187,Y -523.355,Z 327.963,A 0.000,B 0.000,C 90.000,E1 209.283} C_DIS
LIN {X 0.055,Y -518.551,Z 327.952,A 0.000,B 0.000,C 90.000,E1 207.257} C_DIS
LIN {X 0.017,Y -513.929,Z 327.940,A 0.000,B 0.000,C 90.000,E1 205.207} C_DIS
LIN {X 0.027,Y -511.368,Z 327.934,A 0.000,B 0.000,C 90.000,E1 204.027} C_DIS
LIN {X 0.310,Y -508.051,Z 327.925,A 0.000,B 0.000,C 90.000,E1 202.514} C_DIS
LIN {X -0.153,Y -503.401,Z 327.914,A 0.000,B 0.000,C 90.000,E1 200.482} C_DIS
LIN {X 0.066,Y -500.139,Z 327.905,A 0.000,B 0.000,C 90.000,E1 198.960} C_DIS
LIN {X -0.033,Y -496.325,Z 327.895,A 0.000,B 0.000,C 90.000,E1 197.166} C_DIS
LIN {X -0.180,Y -492.111,Z 327.884,A 0.000,B 0.000,C 90.000,E1 195.064} C_DIS
LIN {X -0.116,Y -488.768,Z 327.873,A 0.000,B 0.000,C 90.000,E1 193.231} C_DIS
LIN {X -0.220,Y -486.075,Z 327.865,A 0.000,B 0.000,C 90.000,E1 191.715} C_DIS
LIN {X 0.113,Y -483.432,Z 327.856,A 0.000,B 0.000,C 90.000,E1 190.141} C_DIS
LIN {X -0.088,Y -480.836,Z 327.848,A 0.000,B 0.000,C 90.000,E1 188.624} C_DIS
LIN {X 0.041,Y -476.151,Z 327.831,A 0.000,B 0.000,C 90.000,E1 185.511} C_DIS
LIN {X -0.116,Y -472.786,Z 327.817,A 0.000,B 0.000,C 90.000,E1 183.037} C_DIS
LIN {X -0.005,Y -470.604,Z 327.806,A 0.000,B 0.000,C 90.000,E1 181.146} C_DIS
LIN {X 0.077,Y -467.709,Z 327.789,A 0.000,B 0.000,C 90.000,E1 177.993} C_DIS
LIN {X -0.105,Y -465.729,Z 327.770,A 0.000,B 0.000,C 90.000,E1 174.546} C_DIS
LIN {X -0.232,Y -465.012,Z 327.750,A 0.000,B 0.000,C 90.000,E1 171.084} C_DIS
LIN {X 0.027,Y -465.143,Z 327.736,A 0.000,B 0.000,C 90.000,E1 168.522} C_DIS
LIN {X 0.089,Y -466.165,Z 327.719,A 0.000,B 0.000,C 90.000,E1 165.353} C_DIS
LIN {X 0.169,Y -467.199,Z 327.708,A 0.000,B 0.000,C 90.000,E1 163.449} C_DIS
LIN {X -0.104,Y -470.575,Z 327.685,A 0.000,B 0.000,C 90.000,E1 159.390} C_DIS
LIN {X 0.171,Y -473.955,Z 327.670,A 0.000,B 0.000,C 90.000,E1 156.538} C_DIS
LIN {X -0.085,Y -477.796,Z 327.656,A 0.000,B 0.000,C 90.000,E1 154.076} C_DIS
LIN {X 0.186,Y -482.972,Z 327.641,A 0.000,B 0.000,C 90.000,E1 151.257} C_DIS
LIN {X 0.017,Y -487.596,Z 327.629,A 0.000,B 0.000,C 90.000,E1 149.125} C_DIS
LIN {X 0.144,Y -491.254,Z 327.620,A 0.000,B 0.000,C 90.000,E1 147.582} C_DIS
LIN {X 0.070,Y -494.415,Z 327.613,A 0.000,B 0.000,C 90.000,E1 146.373} C_DIS
LIN {X -0.236,Y -498.440,Z 327.605,A 0.000,B 0.000,C 90.000,E1 144.895} C_DIS
LIN {X 0.008,Y -504.115,Z 327.593,A 0.000,B 0.000,C 90.000,E1 142.763} C_DIS
LIN {X 0.288,Y -507.256,Z 327.587,A 0.000,B 0.000,C 90.000,E1 141.537} C_DIS
LIN {X -0.013,Y -509.375,Z 327.582,A 0.000,B 0.000,C 90.000,E1 140.678} C_DIS
LIN {X 0.269,Y -511.926,Z 327.575,A 0.000,B 0.000,C 90.000,E1 139.461} C_DIS
LIN {X -0.130,Y -514.263,Z 327.568,A 0.000,B 0.000,C 90.000,E1 138.324} C_DIS
LIN {X 0.309,Y -515.732,Z 327.564,A 0.000,B 0.000,C 90.000,E1 137.391} C_DIS
LIN {X 0.034,Y -516.852,Z 327.559,A 0.000,B 0.000,C 90.000,E1 136.539} C_DIS
LIN {X 0.128,Y -517.536,Z 327.554,A 0.000,B 0.000,C 90.000,E1 135.648} C_DIS
LIN {X -0.220,Y -518.027,Z 327.547,A 0.000,B 0.000,C 90.000,E1 134.514} C_DIS
LIN {X -0.112,Y -518.085,Z 327.542,A 0.000,B 0.000,C 90.000,E1 133.623} C_DIS
LIN {X -0.010,Y -517.814,Z 327.537,A 0.000,B 0.000,C 90.000,E1 132.732} C_DIS
LIN {X -0.155,Y -517.526,Z 327.534,A 0.000,B 0.000,C 90.000,E1 132.162} C_DIS
LIN {X -0.065,Y -516.798,Z 327.529,A 0.000,B 0.000,C 90.000,E1 131.272} C_DIS
LIN {X 0.059,Y -515.822,Z 327.524,A 0.000,B 0.000,C 90.000,E1 130.378} C_DIS
LIN {X 0.028,Y -513.909,Z 327.516,A 0.000,B 0.000,C 90.000,E1 128.910} C_DIS
LIN {X -0.116,Y -511.432,Z 327.506,A 0.000,B 0.000,C 90.000,E1 127.156} C_DIS
LIN {X -0.037,Y -509.738,Z 327.500,A 0.000,B 0.000,C 90.000,E1 125.964} C_DIS
LIN {X 0.021,Y -507.767,Z 327.493,A 0.000,B 0.000,C 90.000,E1 124.771} C_DIS
LIN {X 0.046,Y -505.636,Z 327.487,A 0.000,B 0.000,C 90.000,E1 123.579} C_DIS
LIN {X -0.243,Y -503.300,Z 327.480,A 0.000,B 0.000,C 90.000,E1 122.418} C_DIS
LIN {X -0.140,Y -500.863,Z 327.473,A 0.000,B 0.000,C 90.000,E1 121.209} C_DIS
LIN {X 0.211,Y -497.780,Z 327.465,A 0.000,B 0.000,C 90.000,E1 119.667} C_DIS
LIN {X -0.023,Y -495.222,Z 327.458,A 0.000,B 0.000,C 90.000,E1 118.487} C_DIS
LIN {X 0.015,Y -490.655,Z 327.447,A 0.000,B 0.000,C 90.000,E1 116.360} C_DIS
LIN {X -0.108,Y -488.068,Z 327.440,A 0.000,B 0.000,C 90.000,E1 115.155} C_DIS
LIN {X -0.254,Y -484.725,Z 327.431,A 0.000,B 0.000,C 90.000,E1 113.643} C_DIS
LIN {X -0.028,Y -481.271,Z 327.423,A 0.000,B 0.000,C 90.000,E1 112.078} C_DIS
LIN {X -0.225,Y -477.854,Z 327.414,A 0.000,B 0.000,C 90.000,E1 110.556} C_DIS
LIN {X 0.153,Y -474.905,Z 327.407,A 0.000,B 0.000,C 90.000,E1 109.268} C_DIS
LIN {X 0.282,Y -471.153,Z 327.399,A 0.000,B 0.000,C 90.000,E1 107.692} C_DIS
LIN {X -0.141,Y -468.777,Z 327.393,A 0.000,B 0.000,C 90.000,E1 106.804} C_DIS
LIN {X 0.065,Y -465.889,Z 327.387,A 0.000,B 0.000,C 90.000,E1 105.662} C_DIS
LIN {X 0.026,Y -465.879,Z 327.387,A 0.000,B 0.000,C 90.000,E1 105.662} C_DIS
LIN {X -0.021,Y -467.776,Z 327.383,A 0.000,B 0.000,C 90.000,E1 104.898} C_DIS
LIN {X -0.049,Y -475.982,Z 327.357,A 0.000,B 0.000,C 90.000,E1 100.197} C_DIS
LIN {X 0.100,Y -476.685,Z 327.353,A 0.000,B 0.000,C 90.000,E1 99.557} C_DIS
LIN {X -0.254,Y -481.926,Z 327.331,A 0.000,B 0.000,C 90.000,E1 95.568} C_DIS
LIN {X 0.073,Y -482.206,Z 327.329,A 0.000,B 0.000,C 90.000,E1 95.220} C_DIS
LIN {X 0.011,Y -485.398,Z 327.305,A 0.000,B 0.000,C 90.000,E1 90.917} C_DIS
LIN {X -0.165,Y -485.529,Z 327.303,A 0.000,B 0.000,C 90.000,E1 90.630} C_DIS
LIN {X 0.044,Y -486.362,Z 327.281,A 0.000,B 0.000,C 90.000,E1 86.617} C_DIS
LIN {X -0.131,Y -486.367,Z 327.280,A 0.000,B 0.000,C 90.000,E1 86.331} C_DIS
LIN {X -0.142,Y -485.853,Z 327.274,A 0.000,B 0.000,C 90.000,E1 85.412} C_DIS
LIN {X -0.108,Y -484.692,Z 327.254,A 0.000,B 0.000,C 90.000,E1 81.724} C_DIS
LIN {X -0.239,Y -484.496,Z 327.252,A 0.000,B 0.000,C 90.000,E1 81.432} C_DIS
LIN {X 0.099,Y -480.427,Z 327.227,A 0.000,B 0.000,C 90.000,E1 76.769} C_DIS
LIN {X -0.128,Y -477.281,Z 327.215,A 0.000,B 0.000,C 90.000,E1 74.755} C_DIS
LIN {X -0.169,Y -477.282,Z 327.215,A 0.000,B 0.000,C 90.000,E1 74.755} C_DIS
LIN {X -0.020,Y -480.593,Z 327.209,A 0.000,B 0.000,C 90.000,E1 73.685} C_DIS
LIN {X -0.204,Y -483.308,Z 327.204,A 0.000,B 0.000,C 90.000,E1 72.779} C_DIS
LIN {X -0.015,Y -488.337,Z 327.194,A 0.000,B 0.000,C 90.000,E1 70.913} C_DIS
LIN {X -0.049,Y -492.612,Z 327.186,A 0.000,B 0.000,C 90.000,E1 69.390} C_DIS
LIN {X 0.230,Y -497.798,Z 327.175,A 0.000,B 0.000,C 90.000,E1 67.539} C_DIS
LIN {X 0.162,Y -502.921,Z 327.165,A 0.000,B 0.000,C 90.000,E1 65.741} C_DIS
LIN {X -0.142,Y -507.225,Z 327.157,A 0.000,B 0.000,C 90.000,E1 64.280} C_DIS
LIN {X -0.011,Y -510.699,Z 327.150,A 0.000,B 0.000,C 90.000,E1 63.076} C_DIS
LIN {X -0.049,Y -515.825,Z 327.141,A 0.000,B 0.000,C 90.000,E1 61.307} C_DIS
LIN {X 0.106,Y -520.034,Z 327.132,A 0.000,B 0.000,C 90.000,E1 59.822} C_DIS
LIN {X -0.032,Y -524.245,Z 327.124,A 0.000,B 0.000,C 90.000,E1 58.377} C_DIS
LIN {X 0.085,Y -528.441,Z 327.116,A 0.000,B 0.000,C 90.000,E1 56.914} C_DIS
LIN {X 0.099,Y -533.281,Z 327.107,A 0.000,B 0.000,C 90.000,E1 55.182} C_DIS
LIN {X -0.228,Y -537.081,Z 327.099,A 0.000,B 0.000,C 90.000,E1 53.783} C_DIS
LIN {X -0.191,Y -539.888,Z 327.092,A 0.000,B 0.000,C 90.000,E1 52.637} C_DIS
LIN {X 0.246,Y -543.082,Z 327.084,A 0.000,B 0.000,C 90.000,E1 51.170} C_DIS
LIN {X -0.026,Y -545.929,Z 327.077,A 0.000,B 0.000,C 90.000,E1 49.784} C_DIS
LIN {X 0.046,Y -548.394,Z 327.069,A 0.000,B 0.000,C 90.000,E1 48.366} C_DIS
LIN {X -0.195,Y -550.454,Z 327.061,A 0.000,B 0.000,C 90.000,E1 46.986} C_DIS
LIN {X 0.326,Y -551.836,Z 327.055,A 0.000,B 0.000,C 90.000,E1 45.810} C_DIS
LIN {X 0.042,Y -552.634,Z 327.050,A 0.000,B 0.000,C 90.000,E1 45.000} C_DIS
LIN {X 0.196,Y -553.331,Z 327.044,A 0.000,B 0.000,C 90.000,E1 43.866} C_DIS
LIN {X -0.079,Y -553.669,Z 327.039,A 0.000,B 0.000,C 90.000,E1 43.056} C_DIS
LIN {X 0.053,Y -553.830,Z 327.035,A 0.000,B 0.000,C 90.000,E1 42.204} C_DIS
LIN {X -0.241,Y -553.885,Z 327.031,A 0.000,B 0.000,C 90.000,E1 41.676} C_DIS
LIN {X -0.108,Y -553.723,Z 327.027,A 0.000,B 0.000,C 90.000,E1 40.825} C_DIS
LIN {X 0.086,Y -553.374,Z 327.022,A 0.000,B 0.000,C 90.000,E1 39.967} C_DIS
LIN {X 0.274,Y -552.582,Z 327.016,A 0.000,B 0.000,C 90.000,E1 38.830} C_DIS
LIN {X 0.097,Y -551.541,Z 327.010,A 0.000,B 0.000,C 90.000,E1 37.729} C_DIS
LIN {X -0.043,Y -550.162,Z 327.002,A 0.000,B 0.000,C 90.000,E1 36.343} C_DIS
LIN {X -0.146,Y -548.947,Z 326.996,A 0.000,B 0.000,C 90.000,E1 35.231} C_DIS
LIN {X 0.098,Y -546.091,Z 326.982,A 0.000,B 0.000,C 90.000,E1 32.673} C_DIS
LIN {X 0.108,Y -543.847,Z 326.969,A 0.000,B 0.000,C 90.000,E1 30.413} C_DIS
LIN {X 0.056,Y -542.017,Z 326.958,A 0.000,B 0.000,C 90.000,E1 28.437} C_DIS
LIN {X -0.307,Y -540.175,Z 326.947,A 0.000,B 0.000,C 90.000,E1 26.488} C_DIS
LIN {X -0.211,Y -538.612,Z 326.938,A 0.000,B 0.000,C 90.000,E1 24.771} C_DIS
LIN {X 0.056,Y -536.641,Z 326.925,A 0.000,B 0.000,C 90.000,E1 22.461} C_DIS
LIN {X -0.217,Y -534.809,Z 326.909,A 0.000,B 0.000,C 90.000,E1 19.631} C_DIS
LIN {X 0.139,Y -533.922,Z 326.899,A 0.000,B 0.000,C 90.000,E1 17.873} C_DIS
LIN {X 0.054,Y -532.844,Z 326.885,A 0.000,B 0.000,C 90.000,E1 15.300} C_DIS
LIN {X 0.208,Y -532.162,Z 326.869,A 0.000,B 0.000,C 90.000,E1 12.411} C_DIS
LIN {X -0.068,Y -532.168,Z 326.856,A 0.000,B 0.000,C 90.000,E1 10.141} C_DIS
LIN {X 0.104,Y -532.363,Z 326.850,A 0.000,B 0.000,C 90.000,E1 8.973} C_DIS
LIN {X 0.224,Y -533.242,Z 326.834,A 0.000,B 0.000,C 90.000,E1 6.087} C_DIS
LIN {X -0.220,Y -534.921,Z 326.816,A 0.000,B 0.000,C 90.000,E1 2.980} C_DIS
LIN {X -0.199,Y -536.397,Z 326.805,A 0.000,B 0.000,C 90.000,E1 0.974} C_DIS
LIN {X -0.205,Y -540.132,Z 326.783,A 0.000,B 0.000,C 90.000,E1 356.963} C_DIS
LIN {X -0.060,Y -541.806,Z 326.775,A 0.000,B 0.000,C 90.000,E1 355.527} C_DIS
LIN {X -0.178,Y -544.913,Z 326.761,A 0.000,B 0.000,C 90.000,E1 352.989} C_DIS
LIN {X -0.209,Y -549.196,Z 326.748,A 0.000,B 0.000,C 90.000,E1 350.735} C_DIS
LIN {X 0.170,Y -554.526,Z 326.734,A 0.000,B 0.000,C 90.000,E1 348.173} C_DIS
LIN {X 0.140,Y -557.312,Z 326.728,A 0.000,B 0.000,C 90.000,E1 347.061} C_DIS
LIN {X -0.004,Y -559.048,Z 326.725,A 0.000,B 0.000,C 90.000,E1 346.520} C_DIS
LIN {X -0.309,Y -565.259,Z 326.713,A 0.000,B 0.000,C 90.000,E1 344.338} C_DIS
LIN {X 0.228,Y -570.976,Z 326.702,A 0.000,B 0.000,C 90.000,E1 342.362} C_DIS
LIN {X -0.183,Y -575.148,Z 326.695,A 0.000,B 0.000,C 90.000,E1 341.040} C_DIS
LIN {X 0.045,Y -580.151,Z 326.686,A 0.000,B 0.000,C 90.000,E1 339.390} C_DIS
LIN {X -0.124,Y -588.836,Z 326.671,A 0.000,B 0.000,C 90.000,E1 336.719} C_DIS
LIN {X -0.113,Y -596.101,Z 326.659,A 0.000,B 0.000,C 90.000,E1 334.588} C_DIS
LIN {X -0.060,Y -601.768,Z 326.650,A 0.000,B 0.000,C 90.000,E1 332.999} C_DIS
LIN {X -0.040,Y -605.472,Z 326.644,A 0.000,B 0.000,C 90.000,E1 331.948} C_DIS
LIN {X -0.174,Y -614.005,Z 326.631,A 0.000,B 0.000,C 90.000,E1 329.616} C_DIS
LIN {X -0.225,Y -618.819,Z 326.624,A 0.000,B 0.000,C 90.000,E1 328.329} C_DIS
LIN {X 0.035,Y -621.525,Z 326.620,A 0.000,B 0.000,C 90.000,E1 327.533} C_DIS
LIN {X 0.122,Y -625.003,Z 326.614,A 0.000,B 0.000,C 90.000,E1 326.501} C_DIS
LIN {X -0.269,Y -628.982,Z 326.607,A 0.000,B 0.000,C 90.000,E1 325.261} C_DIS
LIN {X 0.281,Y -632.001,Z 326.601,A 0.000,B 0.000,C 90.000,E1 324.196} C_DIS
LIN {X -0.140,Y -635.566,Z 326.594,A 0.000,B 0.000,C 90.000,E1 322.970} C_DIS
LIN {X -0.108,Y -639.790,Z 326.586,A 0.000,B 0.000,C 90.000,E1 321.457} C_DIS
LIN {X -0.179,Y -645.520,Z 326.575,A 0.000,B 0.000,C 90.000,E1 319.461} C_DIS
LIN {X 0.442,Y -649.162,Z 326.568,A 0.000,B 0.000,C 90.000,E1 318.162} C_DIS
LIN {X -0.010,Y -656.648,Z 326.554,A 0.000,B 0.000,C 90.000,E1 315.729} C_DIS
LIN {X -0.130,Y -659.727,Z 326.549,A 0.000,B 0.000,C 90.000,E1 314.757} C_DIS
LIN {X -0.229,Y -663.383,Z 326.542,A 0.000,B 0.000,C 90.000,E1 313.542} C_DIS
LIN {X 0.216,Y -666.162,Z 326.536,A 0.000,B 0.000,C 90.000,E1 312.528} C_DIS
LIN {X -0.245,Y -668.821,Z 326.531,A 0.000,B 0.000,C 90.000,E1 311.595} C_DIS
LIN {X -0.167,Y -671.898,Z 326.524,A 0.000,B 0.000,C 90.000,E1 310.378} C_DIS
LIN {X 0.050,Y -674.762,Z 326.518,A 0.000,B 0.000,C 90.000,E1 309.152} C_DIS
LIN {X -0.340,Y -676.325,Z 326.514,A 0.000,B 0.000,C 90.000,E1 308.463} C_DIS
LIN {X -0.041,Y -678.714,Z 326.507,A 0.000,B 0.000,C 90.000,E1 307.237} C_DIS
LIN {X -0.265,Y -680.313,Z 326.502,A 0.000,B 0.000,C 90.000,E1 306.297} C_DIS
LIN {X -0.087,Y -681.355,Z 326.498,A 0.000,B 0.000,C 90.000,E1 305.564} C_DIS
LIN {X -0.125,Y -682.284,Z 326.492,A 0.000,B 0.000,C 90.000,E1 304.612} C_DIS
LIN {X -0.327,Y -682.779,Z 326.488,A 0.000,B 0.000,C 90.000,E1 303.913} C_DIS
LIN {X -0.335,Y -683.097,Z 326.483,A 0.000,B 0.000,C 90.000,E1 302.959} C_DIS
LIN {X 0.041,Y -682.950,Z 326.479,A 0.000,B 0.000,C 90.000,E1 302.212} C_DIS
LIN {X 0.032,Y -682.336,Z 326.474,A 0.000,B 0.000,C 90.000,E1 301.258} C_DIS
LIN {X 0.047,Y -681.631,Z 326.470,A 0.000,B 0.000,C 90.000,E1 300.541} C_DIS
LIN {X 0.008,Y -680.215,Z 326.464,A 0.000,B 0.000,C 90.000,E1 299.589} C_DIS
LIN {X 0.006,Y -678.902,Z 326.460,A 0.000,B 0.000,C 90.000,E1 298.871} C_DIS
LIN {X 0.183,Y -676.868,Z 326.455,A 0.000,B 0.000,C 90.000,E1 297.897} C_DIS
LIN {X 0.211,Y -674.067,Z 326.448,A 0.000,B 0.000,C 90.000,E1 296.693} C_DIS
LIN {X 0.322,Y -671.631,Z 326.443,A 0.000,B 0.000,C 90.000,E1 295.720} C_DIS
LIN {X -0.298,Y -667.195,Z 326.434,A 0.000,B 0.000,C 90.000,E1 294.079} C_DIS
LIN {X 0.063,Y -663.103,Z 326.426,A 0.000,B 0.000,C 90.000,E1 292.589} C_DIS
LIN {X 0.339,Y -659.003,Z 326.417,A 0.000,B 0.000,C 90.000,E1 291.099} C_DIS
LIN {X 0.291,Y -655.092,Z 326.409,A 0.000,B 0.000,C 90.000,E1 289.631} C_DIS
LIN {X -0.050,Y -651.389,Z 326.401,A 0.000,B 0.000,C 90.000,E1 288.181} C_DIS
LIN {X -0.079,Y -646.232,Z 326.389,A 0.000,B 0.000,C 90.000,E1 285.953} C_DIS
LIN {X -0.161,Y -641.086,Z 326.375,A 0.000,B 0.000,C 90.000,E1 283.467} C_DIS
LIN {X -0.088,Y -635.797,Z 326.357,A 0.000,B 0.000,C 90.000,E1 280.197} C_DIS
LIN {X -0.087,Y -631.892,Z 326.337,A 0.000,B 0.000,C 90.000,E1 276.663} C_DIS
LIN {X 0.180,Y -630.343,Z 326.324,A 0.000,B 0.000,C 90.000,E1 274.359} C_DIS
LIN {X 0.042,Y -629.389,Z 326.310,A 0.000,B 0.000,C 90.000,E1 271.835} C_DIS
LIN {X 0.127,Y -629.198,Z 326.298,A 0.000,B 0.000,C 90.000,E1 269.542} C_DIS
LIN {X -0.146,Y -629.607,Z 326.286,A 0.000,B 0.000,C 90.000,E1 267.535} C_DIS
LIN {X -0.250,Y -630.880,Z 326.272,A 0.000,B 0.000,C 90.000,E1 265.008} C_DIS
LIN {X -0.187,Y -632.740,Z 326.258,A 0.000,B 0.000,C 90.000,E1 262.470} C_DIS
LIN {X 0.010,Y -635.075,Z 326.244,A 0.000,B 0.000,C 90.000,E1 259.926} C_DIS
LIN {X -0.011,Y -638.064,Z 326.230,A 0.000,B 0.000,C 90.000,E1 257.409} C_DIS
LIN {X 0.072,Y -640.492,Z 326.220,A 0.000,B 0.000,C 90.000,E1 255.644} C_DIS
LIN {X 0.376,Y -641.376,Z 326.216,A 0.000,B 0.000,C 90.000,E1 254.866} C_DIS
LIN {X -0.254,Y -642.373,Z 326.211,A 0.000,B 0.000,C 90.000,E1 253.921} C_DIS
LIN {X -0.048,Y -643.340,Z 326.204,A 0.000,B 0.000,C 90.000,E1 252.653} C_DIS
LIN {X 0.139,Y -643.928,Z 326.198,A 0.000,B 0.000,C 90.000,E1 251.638} C_DIS
LIN {X -0.128,Y -644.049,Z 326.194,A 0.000,B 0.000,C 90.000,E1 250.913} C_DIS
LIN {X 0.209,Y -643.943,Z 326.190,A 0.000,B 0.000,C 90.000,E1 250.134} C_DIS
LIN {X 0.158,Y -643.615,Z 326.186,A 0.000,B 0.000,C 90.000,E1 249.390} C_DIS
LIN {X 0.111,Y -642.926,Z 326.181,A 0.000,B 0.000,C 90.000,E1 248.646} C_DIS
LIN {X -0.179,Y -641.913,Z 326.177,A 0.000,B 0.000,C 90.000,E1 247.922} C_DIS
LIN {X -0.243,Y -640.597,Z 326.173,A 0.000,B 0.000,C 90.000,E1 247.177} C_DIS
LIN {X -0.124,Y -639.623,Z 326.170,A 0.000,B 0.000,C 90.000,E1 246.666} C_DIS
LIN {X -0.209,Y -637.909,Z 326.166,A 0.000,B 0.000,C 90.000,E1 245.921} C_DIS
LIN {X -0.266,Y -635.407,Z 326.161,A 0.000,B 0.000,C 90.000,E1 244.921} C_DIS
LIN {X -0.130,Y -633.233,Z 326.156,A 0.000,B 0.000,C 90.000,E1 244.152} C_DIS
LIN {X 0.021,Y -630.026,Z 326.151,A 0.000,B 0.000,C 90.000,E1 243.127} C_DIS
LIN {X 0.143,Y -625.893,Z 326.144,A 0.000,B 0.000,C 90.000,E1 241.847} C_DIS
LIN {X -0.061,Y -620.855,Z 326.135,A 0.000,B 0.000,C 90.000,E1 240.333} C_DIS
LIN {X -0.046,Y -615.747,Z 326.127,A 0.000,B 0.000,C 90.000,E1 238.791} C_DIS
LIN {X -0.087,Y -611.498,Z 326.119,A 0.000,B 0.000,C 90.000,E1 237.502} C_DIS
LIN {X -0.200,Y -607.188,Z 326.112,A 0.000,B 0.000,C 90.000,E1 236.215} C_DIS
LIN {X 0.106,Y -601.043,Z 326.102,A 0.000,B 0.000,C 90.000,E1 234.356} C_DIS
LIN {X -0.234,Y -597.481,Z 326.096,A 0.000,B 0.000,C 90.000,E1 233.336} C_DIS
LIN {X -0.138,Y -593.716,Z 326.090,A 0.000,B 0.000,C 90.000,E1 232.271} C_DIS
LIN {X 0.089,Y -584.479,Z 326.076,A 0.000,B 0.000,C 90.000,E1 229.585} C_DIS
LIN {X -0.312,Y -577.327,Z 326.064,A 0.000,B 0.000,C 90.000,E1 227.472} C_DIS
LIN {X 0.320,Y -572.948,Z 326.056,A 0.000,B 0.000,C 90.000,E1 226.053} C_DIS
LIN {X 0.055,Y -568.404,Z 326.048,A 0.000,B 0.000,C 90.000,E1 224.717} C_DIS
LIN {X -0.189,Y -563.181,Z 326.039,A 0.000,B 0.000,C 90.000,E1 223.095} C_DIS
LIN {X 0.005,Y -556.207,Z 326.027,A 0.000,B 0.000,C 90.000,E1 220.862} C_DIS
LIN {X 0.231,Y -552.710,Z 326.021,A 0.000,B 0.000,C 90.000,E1 219.725} C_DIS
LIN {X -0.267,Y -547.606,Z 326.012,A 0.000,B 0.000,C 90.000,E1 218.096} C_DIS
LIN {X -0.010,Y -542.495,Z 326.002,A 0.000,B 0.000,C 90.000,E1 216.377} C_DIS
LIN {X 0.292,Y -534.609,Z 325.986,A 0.000,B 0.000,C 90.000,E1 213.499} C_DIS
LIN {X -0.236,Y -528.649,Z 325.974,A 0.000,B 0.000,C 90.000,E1 211.258} C_DIS
LIN {X 0.078,Y -524.543,Z 325.964,A 0.000,B 0.000,C 90.000,E1 209.489} C_DIS
LIN {X -0.154,Y -520.358,Z 325.954,A 0.000,B 0.000,C 90.000,E1 207.769} C_DIS
LIN {X -0.144,Y -515.660,Z 325.943,A 0.000,B 0.000,C 90.000,E1 205.720} C_DIS
LIN {X -0.126,Y -511.790,Z 325.933,A 0.000,B 0.000,C 90.000,E1 203.951} C_DIS
LIN {X -0.034,Y -508.476,Z 325.925,A 0.000,B 0.000,C 90.000,E1 202.461} C_DIS
LIN {X -0.005,Y -503.848,Z 325.913,A 0.000,B 0.000,C 90.000,E1 200.375} C_DIS
LIN {X -0.243,Y -500.619,Z 325.905,A 0.000,B 0.000,C 90.000,E1 198.906} C_DIS
LIN {X -0.231,Y -497.489,Z 325.897,A 0.000,B 0.000,C 90.000,E1 197.402} C_DIS
LIN {X -0.075,Y -492.109,Z 325.881,A 0.000,B 0.000,C 90.000,E1 194.662} C_DIS
LIN {X -0.114,Y -488.319,Z 325.870,A 0.000,B 0.000,C 90.000,E1 192.535} C_DIS
LIN {X 0.105,Y -484.634,Z 325.858,A 0.000,B 0.000,C 90.000,E1 190.366} C_DIS
LIN {X 0.184,Y -481.509,Z 325.847,A 0.000,B 0.000,C 90.000,E1 188.511} C_DIS
LIN {X 0.078,Y -477.336,Z 325.832,A 0.000,B 0.000,C 90.000,E1 185.739} C_DIS
LIN {X 0.138,Y -474.351,Z 325.820,A 0.000,B 0.000,C 90.000,E1 183.555} C_DIS
LIN {X -0.133,Y -471.414,Z 325.806,A 0.000,B 0.000,C 90.000,E1 181.088} C_DIS
LIN {X 0.219,Y -468.339,Z 325.787,A 0.000,B 0.000,C 90.000,E1 177.593} C_DIS
LIN {X -0.150,Y -466.418,Z 325.766,A 0.000,B 0.000,C 90.000,E1 173.856} C_DIS
LIN {X 0.075,Y -465.902,Z 325.745,A 0.000,B 0.000,C 90.000,E1 170.038} C_DIS
LIN {X 0.069,Y -466.430,Z 325.727,A 0.000,B 0.000,C 90.000,E1 166.881} C_DIS
LIN {X 0.026,Y -467.771,Z 325.711,A 0.000,B 0.000,C 90.000,E1 164.047} C_DIS
LIN {X -0.028,Y -471.445,Z 325.685,A 0.000,B 0.000,C 90.000,E1 159.337} C_DIS
LIN {X -0.166,Y -474.805,Z 325.670,A 0.000,B 0.000,C 90.000,E1 156.538} C_DIS
LIN {X 0.009,Y -479.105,Z 325.654,A 0.000,B 0.000,C 90.000,E1 153.717} C_DIS
LIN {X -0.090,Y -483.090,Z 325.642,A 0.000,B 0.000,C 90.000,E1 151.563} C_DIS
LIN {X 0.225,Y -489.622,Z 325.625,A 0.000,B 0.000,C 90.000,E1 148.456} C_DIS
LIN {X 0.085,Y -494.945,Z 325.613,A 0.000,B 0.000,C 90.000,E1 146.342} C_DIS
LIN {X -0.049,Y -500.403,Z 325.601,A 0.000,B 0.000,C 90.000,E1 144.242} C_DIS
LIN {X 0.052,Y -505.107,Z 325.591,A 0.000,B 0.000,C 90.000,E1 142.431} C_DIS
LIN {X 0.044,Y -507.325,Z 325.586,A 0.000,B 0.000,C 90.000,E1 141.537} C_DIS
LIN {X 0.066,Y -509.322,Z 325.581,A 0.000,B 0.000,C 90.000,E1 140.642} C_DIS
LIN {X 0.022,Y -511.784,Z 325.575,A 0.000,B 0.000,C 90.000,E1 139.461} C_DIS
LIN {X -0.037,Y -514.004,Z 325.568,A 0.000,B 0.000,C 90.000,E1 138.286} C_DIS
LIN {X 0.055,Y -515.373,Z 325.563,A 0.000,B 0.000,C 90.000,E1 137.391} C_DIS
LIN {X -0.223,Y -516.434,Z 325.558,A 0.000,B 0.000,C 90.000,E1 136.539} C_DIS
LIN {X -0.134,Y -517.097,Z 325.554,A 0.000,B 0.000,C 90.000,E1 135.648} C_DIS
LIN {X 0.243,Y -517.526,Z 325.547,A 0.000,B 0.000,C 90.000,E1 134.433} C_DIS
LIN {X -0.109,Y -517.486,Z 325.541,A 0.000,B 0.000,C 90.000,E1 133.299} C_DIS
LIN {X 0.016,Y -517.104,Z 325.536,A 0.000,B 0.000,C 90.000,E1 132.405} C_DIS
LIN {X 0.105,Y -516.412,Z 325.531,A 0.000,B 0.000,C 90.000,E1 131.515} C_DIS
LIN {X 0.226,Y -515.498,Z 325.526,A 0.000,B 0.000,C 90.000,E1 130.620} C_DIS
LIN {X -0.283,Y -513.171,Z 325.516,A 0.000,B 0.000,C 90.000,E1 128.910} C_DIS
LIN {X -0.276,Y -511.488,Z 325.509,A 0.000,B 0.000,C 90.000,E1 127.729} C_DIS
LIN {X 0.016,Y -509.421,Z 325.501,A 0.000,B 0.000,C 90.000,E1 126.217} C_DIS
LIN {X 0.156,Y -508.010,Z 325.496,A 0.000,B 0.000,C 90.000,E1 125.311} C_DIS
LIN {X 0.077,Y -505.384,Z 325.488,A 0.000,B 0.000,C 90.000,E1 123.833} C_DIS
LIN {X 0.202,Y -503.096,Z 325.481,A 0.000,B 0.000,C 90.000,E1 122.625} C_DIS
LIN {X 0.037,Y -499.434,Z 325.471,A 0.000,B 0.000,C 90.000,E1 120.846} C_DIS
LIN {X 0.103,Y -496.335,Z 325.463,A 0.000,B 0.000,C 90.000,E1 119.333} C_DIS
LIN {X -0.154,Y -493.752,Z 325.456,A 0.000,B 0.000,C 90.000,E1 118.153} C_DIS
LIN {X -0.160,Y -489.281,Z 325.445,A 0.000,B 0.000,C 90.000,E1 116.027} C_DIS
LIN {X 0.153,Y -486.035,Z 325.436,A 0.000,B 0.000,C 90.000,E1 114.463} C_DIS
LIN {X -0.036,Y -482.680,Z 325.428,A 0.000,B 0.000,C 90.000,E1 112.950} C_DIS
LIN {X -0.052,Y -477.971,Z 325.416,A 0.000,B 0.000,C 90.000,E1 110.791} C_DIS
LIN {X -0.101,Y -475.898,Z 325.410,A 0.000,B 0.000,C 90.000,E1 109.866} C_DIS
LIN {X -0.184,Y -470.788,Z 325.398,A 0.000,B 0.000,C 90.000,E1 107.692} C_DIS
LIN {X 0.170,Y -466.994,Z 325.389,A 0.000,B 0.000,C 90.000,E1 106.079} C_DIS
LIN {X 0.037,Y -465.881,Z 325.387,A 0.000,B 0.000,C 90.000,E1 105.662} C_DIS
LIN {X -0.003,Y -465.887,Z 325.387,A 0.000,B 0.000,C 90.000,E1 105.662} C_DIS
LIN {X 0.082,Y -467.884,Z 325.382,A 0.000,B 0.000,C 90.000,E1 104.828} C_DIS
LIN {X 0.110,Y -475.447,Z 325.358,A 0.000,B 0.000,C 90.000,E1 100.433} C_DIS
LIN {X -0.053,Y -476.097,Z 325.356,A 0.000,B 0.000,C 90.000,E1 100.141} C_DIS
LIN {X -0.248,Y -482.017,Z 325.331,A 0.000,B 0.000,C 90.000,E1 95.511} C_DIS
LIN {X 0.022,Y -482.684,Z 325.324,A 0.000,B 0.000,C 90.000,E1 94.245} C_DIS
LIN {X 0.022,Y -485.458,Z 325.305,A 0.000,B 0.000,C 90.000,E1 90.859} C_DIS
LIN {X -0.014,Y -485.500,Z 325.300,A 0.000,B 0.000,C 90.000,E1 89.943} C_DIS
LIN {X 0.055,Y -486.383,Z 325.281,A 0.000,B 0.000,C 90.000,E1 86.560} C_DIS
LIN {X -0.121,Y -486.364,Z 325.279,A 0.000,B 0.000,C 90.000,E1 86.274} C_DIS
LIN {X -0.032,Y -484.690,Z 325.254,A 0.000,B 0.000,C 90.000,E1 81.659} C_DIS
LIN {X 0.113,Y -484.064,Z 325.250,A 0.000,B 0.000,C 90.000,E1 81.027} C_DIS
LIN {X -0.231,Y -480.635,Z 325.228,A 0.000,B 0.000,C 90.000,E1 77.061} C_DIS
LIN {X 0.203,Y -480.331,Z 325.226,A 0.000,B 0.000,C 90.000,E1 76.700} C_DIS
LIN {X 0.164,Y -477.157,Z 325.215,A 0.000,B 0.000,C 90.000,E1 74.629} C_DIS
LIN {X 0.124,Y -477.155,Z 325.215,A 0.000,B 0.000,C 90.000,E1 74.629} C_DIS
LIN {X -0.214,Y -479.967,Z 325.210,A 0.000,B 0.000,C 90.000,E1 73.740} C_DIS
LIN {X 0.057,Y -482.665,Z 325.204,A 0.000,B 0.000,C 90.000,E1 72.779} C_DIS
LIN {X 0.233,Y -487.637,Z 325.194,A 0.000,B 0.000,C 90.000,E1 70.913} C_DIS
LIN {X 0.187,Y -491.864,Z 325.186,A 0.000,B 0.000,C 90.000,E1 69.390} C_DIS
LIN {X 0.048,Y -497.848,Z 325.174,A 0.000,B 0.000,C 90.000,E1 67.283} C_DIS
LIN {X -0.090,Y -502.163,Z 325.165,A 0.000,B 0.000,C 90.000,E1 65.793} C_DIS
LIN {X -0.010,Y -508.162,Z 325.154,A 0.000,B 0.000,C 90.000,E1 63.691} C_DIS
LIN {X -0.219,Y -512.463,Z 325.146,A 0.000,B 0.000,C 90.000,E1 62.231} C_DIS
LIN {X 0.128,Y -516.758,Z 325.137,A 0.000,B 0.000,C 90.000,E1 60.717} C_DIS
LIN {X 0.166,Y -522.692,Z 325.126,A 0.000,B 0.000,C 90.000,E1 58.663} C_DIS
LIN {X 0.212,Y -527.695,Z 325.116,A 0.000,B 0.000,C 90.000,E1 56.914} C_DIS
LIN {X 0.213,Y -532.561,Z 325.107,A 0.000,B 0.000,C 90.000,E1 55.182} C_DIS
LIN {X -0.127,Y -535.672,Z 325.100,A 0.000,B 0.000,C 90.000,E1 54.069} C_DIS
LIN {X -0.110,Y -538.518,Z 325.094,A 0.000,B 0.000,C 90.000,E1 52.924} C_DIS
LIN {X 0.303,Y -541.785,Z 325.086,A 0.000,B 0.000,C 90.000,E1 51.457} C_DIS
LIN {X -0.016,Y -544.144,Z 325.080,A 0.000,B 0.000,C 90.000,E1 50.356} C_DIS
LIN {X 0.012,Y -545.783,Z 325.075,A 0.000,B 0.000,C 90.000,E1 49.504} C_DIS
LIN {X -0.262,Y -547.759,Z 325.069,A 0.000,B 0.000,C 90.000,E1 48.405} C_DIS
LIN {X 0.216,Y -549.441,Z 325.063,A 0.000,B 0.000,C 90.000,E1 47.229} C_DIS
LIN {X -0.057,Y -550.931,Z 325.056,A 0.000,B 0.000,C 90.000,E1 46.134} C_DIS
LIN {X 0.073,Y -552.066,Z 325.050,A 0.000,B 0.000,C 90.000,E1 45.000} C_DIS
LIN {X 0.219,Y -552.791,Z 325.044,A 0.000,B 0.000,C 90.000,E1 43.866} C_DIS
LIN {X -0.086,Y -553.099,Z 325.041,A 0.000,B 0.000,C 90.000,E1 43.338} C_DIS
LIN {X 0.065,Y -553.353,Z 325.035,A 0.000,B 0.000,C 90.000,E1 42.204} C_DIS
LIN {X -0.233,Y -553.451,Z 325.031,A 0.000,B 0.000,C 90.000,E1 41.676} C_DIS
LIN {X -0.043,Y -553.254,Z 325.025,A 0.000,B 0.000,C 90.000,E1 40.539} C_DIS
LIN {X -0.274,Y -552.900,Z 325.021,A 0.000,B 0.000,C 90.000,E1 39.725} C_DIS
LIN {X -0.098,Y -552.142,Z 325.014,A 0.000,B 0.000,C 90.000,E1 38.588} C_DIS
LIN {X 0.213,Y -550.923,Z 325.007,A 0.000,B 0.000,C 90.000,E1 37.156} C_DIS
LIN {X -0.264,Y -549.499,Z 324.999,A 0.000,B 0.000,C 90.000,E1 35.804} C_DIS
LIN {X -0.319,Y -547.917,Z 324.991,A 0.000,B 0.000,C 90.000,E1 34.405} C_DIS
LIN {X -0.139,Y -545.565,Z 324.978,A 0.000,B 0.000,C 90.000,E1 32.133} C_DIS
LIN {X 0.114,Y -543.620,Z 324.967,A 0.000,B 0.000,C 90.000,E1 30.129} C_DIS
LIN {X 0.047,Y -542.103,Z 324.958,A 0.000,B 0.000,C 90.000,E1 28.437} C_DIS
LIN {X 0.171,Y -540.263,Z 324.947,A 0.000,B 0.000,C 90.000,E1 26.437} C_DIS
LIN {X -0.216,Y -538.701,Z 324.938,A 0.000,B 0.000,C 90.000,E1 24.771} C_DIS
LIN {X -0.162,Y -536.973,Z 324.926,A 0.000,B 0.000,C 90.000,E1 22.770} C_DIS
LIN {X 0.057,Y -535.219,Z 324.912,A 0.000,B 0.000,C 90.000,E1 20.174} C_DIS
LIN {X -0.054,Y -534.159,Z 324.901,A 0.000,B 0.000,C 90.000,E1 18.181} C_DIS
LIN {X 0.062,Y -532.937,Z 324.885,A 0.000,B 0.000,C 90.000,E1 15.300} C_DIS
LIN {X 0.015,Y -532.292,Z 324.872,A 0.000,B 0.000,C 90.000,E1 13.008} C_DIS
LIN {X -0.216,Y -532.156,Z 324.866,A 0.000,B 0.000,C 90.000,E1 11.883} C_DIS
LIN {X 0.032,Y -532.302,Z 324.853,A 0.000,B 0.000,C 90.000,E1 9.557} C_DIS
LIN {X 0.209,Y -532.733,Z 324.840,A 0.000,B 0.000,C 90.000,E1 7.239} C_DIS
LIN {X -0.277,Y -533.387,Z 324.831,A 0.000,B 0.000,C 90.000,E1 5.568} C_DIS
LIN {X -0.212,Y -534.796,Z 324.816,A 0.000,B 0.000,C 90.000,E1 2.980} C_DIS
LIN {X -0.195,Y -536.178,Z 324.805,A 0.000,B 0.000,C 90.000,E1 0.974} C_DIS
LIN {X -0.216,Y -539.757,Z 324.783,A 0.000,B 0.000,C 90.000,E1 356.963} C_DIS
LIN {X -0.078,Y -541.368,Z 324.775,A 0.000,B 0.000,C 90.000,E1 355.527} C_DIS
LIN {X -0.211,Y -544.415,Z 324.761,A 0.000,B 0.000,C 90.000,E1 352.989} C_DIS
LIN {X -0.157,Y -549.188,Z 324.747,A 0.000,B 0.000,C 90.000,E1 350.443} C_DIS
LIN {X 0.103,Y -553.928,Z 324.734,A 0.000,B 0.000,C 90.000,E1 348.173} C_DIS
LIN {X -0.065,Y -556.027,Z 324.730,A 0.000,B 0.000,C 90.000,E1 347.353} C_DIS
LIN {X 0.064,Y -556.702,Z 324.728,A 0.000,B 0.000,C 90.000,E1 347.061} C_DIS
LIN {X -0.085,Y -558.414,Z 324.725,A 0.000,B 0.000,C 90.000,E1 346.520} C_DIS
LIN {X 0.134,Y -564.610,Z 324.713,A 0.000,B 0.000,C 90.000,E1 344.283} C_DIS
LIN {X 0.111,Y -570.315,Z 324.702,A 0.000,B 0.000,C 90.000,E1 342.362} C_DIS
LIN {X -0.313,Y -574.478,Z 324.695,A 0.000,B 0.000,C 90.000,E1 341.040} C_DIS
LIN {X -0.100,Y -579.470,Z 324.685,A 0.000,B 0.000,C 90.000,E1 339.390} C_DIS
LIN {X 0.245,Y -588.163,Z 324.671,A 0.000,B 0.000,C 90.000,E1 336.666} C_DIS
LIN {X 0.233,Y -595.434,Z 324.659,A 0.000,B 0.000,C 90.000,E1 334.537} C_DIS
LIN {X -0.267,Y -601.106,Z 324.650,A 0.000,B 0.000,C 90.000,E1 332.999} C_DIS
LIN {X 0.276,Y -604.815,Z 324.644,A 0.000,B 0.000,C 90.000,E1 331.897} C_DIS
LIN {X -0.104,Y -613.333,Z 324.631,A 0.000,B 0.000,C 90.000,E1 329.587} C_DIS
LIN {X 0.046,Y -618.146,Z 324.624,A 0.000,B 0.000,C 90.000,E1 328.280} C_DIS
LIN {X -0.228,Y -620.863,Z 324.620,A 0.000,B 0.000,C 90.000,E1 327.533} C_DIS
LIN {X -0.152,Y -624.334,Z 324.614,A 0.000,B 0.000,C 90.000,E1 326.501} C_DIS
LIN {X 0.320,Y -628.337,Z 324.607,A 0.000,B 0.000,C 90.000,E1 325.182} C_DIS
LIN {X -0.016,Y -631.382,Z 324.601,A 0.000,B 0.000,C 90.000,E1 324.196} C_DIS
LIN {X 0.058,Y -634.958,Z 324.594,A 0.000,B 0.000,C 90.000,E1 322.924} C_DIS
LIN {X 0.069,Y -639.189,Z 324.586,A 0.000,B 0.000,C 90.000,E1 321.412} C_DIS
LIN {X 0.390,Y -644.930,Z 324.575,A 0.000,B 0.000,C 90.000,E1 319.380} C_DIS
LIN {X 0.089,Y -648.562,Z 324.568,A 0.000,B 0.000,C 90.000,E1 318.162} C_DIS
LIN {X -0.347,Y -655.289,Z 324.555,A 0.000,B 0.000,C 90.000,E1 315.972} C_DIS
LIN {X -0.022,Y -658.401,Z 324.550,A 0.000,B 0.000,C 90.000,E1 314.960} C_DIS
LIN {X 0.311,Y -662.762,Z 324.542,A 0.000,B 0.000,C 90.000,E1 313.461} C_DIS
LIN {X -0.192,Y -665.530,Z 324.536,A 0.000,B 0.000,C 90.000,E1 312.528} C_DIS
LIN {X 0.280,Y -668.148,Z 324.531,A 0.000,B 0.000,C 90.000,E1 311.515} C_DIS
LIN {X -0.086,Y -671.203,Z 324.524,A 0.000,B 0.000,C 90.000,E1 310.334} C_DIS
LIN {X 0.030,Y -674.043,Z 324.517,A 0.000,B 0.000,C 90.000,E1 309.116} C_DIS
LIN {X 0.158,Y -675.582,Z 324.513,A 0.000,B 0.000,C 90.000,E1 308.382} C_DIS
LIN {X -0.097,Y -677.935,Z 324.507,A 0.000,B 0.000,C 90.000,E1 307.202} C_DIS
LIN {X 0.208,Y -679.491,Z 324.501,A 0.000,B 0.000,C 90.000,E1 306.217} C_DIS
LIN {X -0.019,Y -680.505,Z 324.497,A 0.000,B 0.000,C 90.000,E1 305.518} C_DIS
LIN {X 0.325,Y -681.397,Z 324.492,A 0.000,B 0.000,C 90.000,E1 304.532} C_DIS
LIN {X 0.118,Y -681.721,Z 324.489,A 0.000,B 0.000,C 90.000,E1 304.072} C_DIS
LIN {X -0.087,Y -682.002,Z 324.485,A 0.000,B 0.000,C 90.000,E1 303.372} C_DIS
LIN {X 0.281,Y -682.041,Z 324.481,A 0.000,B 0.000,C 90.000,E1 302.625} C_DIS
LIN {X 0.090,Y -681.887,Z 324.479,A 0.000,B 0.000,C 90.000,E1 302.163} C_DIS
LIN {X 0.074,Y -681.253,Z 324.473,A 0.000,B 0.000,C 90.000,E1 301.209} C_DIS
LIN {X -0.158,Y -680.474,Z 324.469,A 0.000,B 0.000,C 90.000,E1 300.512} C_DIS
LIN {X -0.160,Y -679.413,Z 324.466,A 0.000,B 0.000,C 90.000,E1 299.795} C_DIS
LIN {X -0.168,Y -678.113,Z 324.462,A 0.000,B 0.000,C 90.000,E1 299.077} C_DIS
LIN {X 0.002,Y -676.113,Z 324.456,A 0.000,B 0.000,C 90.000,E1 298.103} C_DIS
LIN {X 0.327,Y -673.314,Z 324.449,A 0.000,B 0.000,C 90.000,E1 296.873} C_DIS
LIN {X 0.132,Y -670.901,Z 324.444,A 0.000,B 0.000,C 90.000,E1 295.924} C_DIS
LIN {X -0.069,Y -665.774,Z 324.433,A 0.000,B 0.000,C 90.000,E1 294.003} C_DIS
LIN {X 0.133,Y -661.026,Z 324.424,A 0.000,B 0.000,C 90.000,E1 292.280} C_DIS
LIN {X 0.218,Y -654.980,Z 324.412,A 0.000,B 0.000,C 90.000,E1 290.066} C_DIS
LIN {X -0.042,Y -650.597,Z 324.402,A 0.000,B 0.000,C 90.000,E1 288.362} C_DIS
LIN {X 0.011,Y -646.501,Z 324.392,A 0.000,B 0.000,C 90.000,E1 286.622} C_DIS
LIN {X -0.206,Y -642.690,Z 324.383,A 0.000,B 0.000,C 90.000,E1 284.898} C_DIS
LIN {X 0.105,Y -639.254,Z 324.373,A 0.000,B 0.000,C 90.000,E1 283.119} C_DIS
LIN {X -0.036,Y -634.860,Z 324.358,A 0.000,B 0.000,C 90.000,E1 280.366} C_DIS
LIN {X 0.244,Y -630.638,Z 324.337,A 0.000,B 0.000,C 90.000,E1 276.549} C_DIS
LIN {X -0.035,Y -628.883,Z 324.321,A 0.000,B 0.000,C 90.000,E1 273.784} C_DIS
LIN {X 0.320,Y -628.169,Z 324.310,A 0.000,B 0.000,C 90.000,E1 271.718} C_DIS
LIN {X -0.002,Y -628.028,Z 324.298,A 0.000,B 0.000,C 90.000,E1 269.714} C_DIS
LIN {X 0.046,Y -628.450,Z 324.286,A 0.000,B 0.000,C 90.000,E1 267.421} C_DIS
LIN {X 0.180,Y -629.628,Z 324.273,A 0.000,B 0.000,C 90.000,E1 265.122} C_DIS
LIN {X -0.132,Y -630.622,Z 324.265,A 0.000,B 0.000,C 90.000,E1 263.628} C_DIS
LIN {X 0.056,Y -632.140,Z 324.255,A 0.000,B 0.000,C 90.000,E1 261.837} C_DIS
LIN {X 0.002,Y -634.416,Z 324.242,A 0.000,B 0.000,C 90.000,E1 259.567} C_DIS
LIN {X -0.161,Y -637.540,Z 324.228,A 0.000,B 0.000,C 90.000,E1 257.061} C_DIS
LIN {X 0.225,Y -639.632,Z 324.220,A 0.000,B 0.000,C 90.000,E1 255.519} C_DIS
LIN {X -0.262,Y -640.544,Z 324.216,A 0.000,B 0.000,C 90.000,E1 254.810} C_DIS
LIN {X -0.112,Y -641.541,Z 324.210,A 0.000,B 0.000,C 90.000,E1 253.795} C_DIS
LIN {X -0.105,Y -642.550,Z 324.203,A 0.000,B 0.000,C 90.000,E1 252.543} C_DIS
LIN {X 0.225,Y -643.041,Z 324.199,A 0.000,B 0.000,C 90.000,E1 251.764} C_DIS
LIN {X -0.053,Y -643.262,Z 324.195,A 0.000,B 0.000,C 90.000,E1 251.040} C_DIS
LIN {X -0.168,Y -643.300,Z 324.192,A 0.000,B 0.000,C 90.000,E1 250.550} C_DIS
LIN {X 0.213,Y -642.935,Z 324.186,A 0.000,B 0.000,C 90.000,E1 249.518} C_DIS
LIN {X 0.269,Y -642.832,Z 324.185,A 0.000,B 0.000,C 90.000,E1 249.263} C_DIS
LIN {X -0.018,Y -642.134,Z 324.181,A 0.000,B 0.000,C 90.000,E1 248.539} C_DIS
LIN {X 0.101,Y -641.562,Z 324.178,A 0.000,B 0.000,C 90.000,E1 248.028} C_DIS
LIN {X -0.151,Y -639.928,Z 324.172,A 0.000,B 0.000,C 90.000,E1 247.050} C_DIS
LIN {X -0.179,Y -637.936,Z 324.167,A 0.000,B 0.000,C 90.000,E1 246.049} C_DIS
LIN {X -0.190,Y -634.932,Z 324.160,A 0.000,B 0.000,C 90.000,E1 244.793} C_DIS
LIN {X -0.058,Y -632.787,Z 324.156,A 0.000,B 0.000,C 90.000,E1 244.024} C_DIS
LIN {X 0.115,Y -628.821,Z 324.149,A 0.000,B 0.000,C 90.000,E1 242.743} C_DIS
LIN {X -0.326,Y -623.914,Z 324.140,A 0.000,B 0.000,C 90.000,E1 241.257} C_DIS
LIN {X -0.018,Y -619.772,Z 324.133,A 0.000,B 0.000,C 90.000,E1 239.950} C_DIS
LIN {X 0.261,Y -613.935,Z 324.123,A 0.000,B 0.000,C 90.000,E1 238.122} C_DIS
LIN {X 0.185,Y -609.694,Z 324.116,A 0.000,B 0.000,C 90.000,E1 236.834} C_DIS
LIN {X 0.103,Y -606.263,Z 324.110,A 0.000,B 0.000,C 90.000,E1 235.801} C_DIS
LIN {X -0.006,Y -601.109,Z 324.101,A 0.000,B 0.000,C 90.000,E1 234.242} C_DIS
LIN {X -0.212,Y -597.538,Z 324.096,A 0.000,B 0.000,C 90.000,E1 233.210} C_DIS
LIN {X -0.365,Y -592.827,Z 324.088,A 0.000,B 0.000,C 90.000,E1 231.904} C_DIS
LIN {X -0.090,Y -585.486,Z 324.076,A 0.000,B 0.000,C 90.000,E1 229.747} C_DIS
LIN {X 0.076,Y -577.449,Z 324.063,A 0.000,B 0.000,C 90.000,E1 227.310} C_DIS
LIN {X -0.101,Y -573.076,Z 324.055,A 0.000,B 0.000,C 90.000,E1 225.972} C_DIS
LIN {X -0.069,Y -565.890,Z 324.043,A 0.000,B 0.000,C 90.000,E1 223.785} C_DIS
LIN {X -0.121,Y -562.426,Z 324.037,A 0.000,B 0.000,C 90.000,E1 222.690} C_DIS
LIN {X -0.035,Y -556.351,Z 324.026,A 0.000,B 0.000,C 90.000,E1 220.744} C_DIS
LIN {X -0.167,Y -552.838,Z 324.020,A 0.000,B 0.000,C 90.000,E1 219.644} C_DIS
LIN {X 0.107,Y -547.739,Z 324.011,A 0.000,B 0.000,C 90.000,E1 217.935} C_DIS
LIN {X 0.000,Y -543.511,Z 324.003,A 0.000,B 0.000,C 90.000,E1 216.537} C_DIS
LIN {X -0.095,Y -535.554,Z 323.987,A 0.000,B 0.000,C 90.000,E1 213.706} C_DIS
LIN {X 0.162,Y -530.301,Z 323.976,A 0.000,B 0.000,C 90.000,E1 211.671} C_DIS
LIN {X 0.009,Y -525.439,Z 323.965,A 0.000,B 0.000,C 90.000,E1 209.667} C_DIS
LIN {X 0.249,Y -521.265,Z 323.955,A 0.000,B 0.000,C 90.000,E1 207.897} C_DIS
LIN {X 0.277,Y -516.519,Z 323.944,A 0.000,B 0.000,C 90.000,E1 205.848} C_DIS
LIN {X -0.154,Y -512.677,Z 323.934,A 0.000,B 0.000,C 90.000,E1 204.131} C_DIS
LIN {X -0.051,Y -509.371,Z 323.926,A 0.000,B 0.000,C 90.000,E1 202.642} C_DIS
LIN {X -0.096,Y -505.351,Z 323.916,A 0.000,B 0.000,C 90.000,E1 200.865} C_DIS
LIN {X -0.304,Y -502.148,Z 323.908,A 0.000,B 0.000,C 90.000,E1 199.396} C_DIS
LIN {X -0.197,Y -498.344,Z 323.898,A 0.000,B 0.000,C 90.000,E1 197.583} C_DIS
LIN {X 0.115,Y -492.943,Z 323.883,A 0.000,B 0.000,C 90.000,E1 194.828} C_DIS
LIN {X -0.022,Y -489.146,Z 323.871,A 0.000,B 0.000,C 90.000,E1 192.715} C_DIS
LIN {X -0.130,Y -485.994,Z 323.860,A 0.000,B 0.000,C 90.000,E1 190.894} C_DIS
LIN {X -0.147,Y -482.389,Z 323.849,A 0.000,B 0.000,C 90.000,E1 188.746} C_DIS
LIN {X 0.109,Y -477.798,Z 323.831,A 0.000,B 0.000,C 90.000,E1 185.625} C_DIS
LIN {X 0.183,Y -474.880,Z 323.819,A 0.000,B 0.000,C 90.000,E1 183.440} C_DIS
LIN {X 0.148,Y -472.362,Z 323.807,A 0.000,B 0.000,C 90.000,E1 181.260} C_DIS
LIN {X -0.159,Y -469.047,Z 323.786,A 0.000,B 0.000,C 90.000,E1 177.535} C_DIS
LIN {X -0.033,Y -467.197,Z 323.765,A 0.000,B 0.000,C 90.000,E1 173.742} C_DIS
LIN {X -0.046,Y -466.699,Z 323.746,A 0.000,B 0.000,C 90.000,E1 170.274} C_DIS
LIN {X 0.162,Y -467.095,Z 323.730,A 0.000,B 0.000,C 90.000,E1 167.409} C_DIS
LIN {X 0.149,Y -468.228,Z 323.714,A 0.000,B 0.000,C 90.000,E1 164.574} C_DIS
END
